# B&R Automation Studio project AriesV2 (part 4)

#### Cyclic.st
```iecst
PROGRAM _CYCLIC

	gRecCfg;
//
//	CASE gHmi.prv.currentPage OF
//		HMI_RECIPE_20_SELECT:
//			pRecCfgUIConnect ACCESS ADR(gRecipe_CSV_UIConnect);
//			pCmd ACCESS ADR(loc.Rec.HMI);
//		HMI_RECIPE_21_PVLIST:
//			pRecCfgUIConnect ACCESS ADR(gRecipe_CSV_UIConnect);
//			pCmd ACCESS ADR(loc.Rec.HMI);
//		HMI_CONFIG_30_SELECT:
//			pRecCfgUIConnect ACCESS ADR(gConfig_CSV_UIConnect);
//			pCmd ACCESS ADR(loc.Cfg.HMI);
//		HMI_CONFIG_31_PVLIST:
//			pRecCfgUIConnect ACCESS ADR(gConfig_CSV_UIConnect);
//			pCmd ACCESS ADR(loc.Cfg.HMI);
//		HMI_LOGIN_43_ENGINEER:
//			pRecCfgUIConnect ACCESS ADR(gConfig_CSV_UIConnect);
//			pCmd ACCESS ADR(loc.Cfg.HMI);
//	END_CASE;
//
//
//	IF EDGENEG(gHmi.prv.currentPage = HMI_RECIPE_20_SELECT) THEN
//		locFindActiveRecipe := 1;
//	END_IF;
//
//	IF EDGENEG(gHmi.prv.currentPage = HMI_CONFIG_30_SELECT) THEN
//		locFindActiveRecipe := 1;
//	END_IF;
//
//	IF loc.Rec.cmd.Copy_default_to_save = 1 THEN
//		gRecCfg.save.Rec := gRecCfg.defaultvals.Rec;
//	END_IF;
//
//	IF loc.Rec.cmd.Copy_default_to_active = 1 THEN
//		gRecCfg.active.Rec := gRecCfg.defaultvals.Rec;
//	END_IF;
//
//	IF loc.Rec.cmd.Copy_save_to_active = 1 THEN
//		gRecCfg.active.Rec := gRecCfg.save.Rec;
//	END_IF;
//
//	IF loc.Rec.cmd.Copy_save_to_default = 1 THEN
//		gRecCfg.defaultvals.Rec := gRecCfg.save.Rec;
//	END_IF;
//
//	IF loc.Rec.cmd.Copy_active_to_save = 1 THEN
//		gRecCfg.save.Rec := gRecCfg.active.Rec;
//	END_IF;
//
//	IF loc.Rec.cmd.Copy_active_to_default = 1 THEN
//		gRecCfg.defaultvals.Rec := gRecCfg.active.Rec;
//	END_IF;
//
//	IF loc.Rec.cmd.Copy_internal_to_default = 1 THEN
////		Set_Default_Rec;
//	END_IF;
//
//	gRecCfg.save.Cfg.Motor.Home := gRecCfg.active.Cfg.Motor.Home;
//
//	loc.Cfg.status.save_differs_from_active := BOOL_TO_USINT(brsmemcmp(ADR(gRecCfg.save.Cfg),ADR(gRecCfg.active.Cfg), SIZEOF(Global_Cfg_typ)) <> 0);
//	loc.Cfg.status.default_differs_from_save := BOOL_TO_USINT(brsmemcmp(ADR(gRecCfg.defaultvals.Cfg),ADR(gRecCfg.save.Cfg), SIZEOF(Global_Cfg_typ)) <> 0);
//	loc.Cfg.status.active_differs_from_default := BOOL_TO_USINT(brsmemcmp(ADR(gRecCfg.active.Cfg),ADR(gRecCfg.defaultvals.Cfg), SIZEOF(Global_Cfg_typ)) <> 0);
//
////	loc.Cfg.status.Invalid := NOT Fcn_Config_Valid(pCfg := ADR(gRecCfg.active.Cfg), pAlarms := ADR(gAlarms));
//
//	loc.Rec.status.save_differs_from_active := BOOL_TO_USINT(brsmemcmp(ADR(gRecCfg.save.Rec),ADR(gRecCfg.active.Rec), SIZEOF(Global_Rec_typ)) <> 0);
//	loc.Rec.status.default_differs_from_save := BOOL_TO_USINT(brsmemcmp(ADR(gRecCfg.defaultvals.Rec),ADR(gRecCfg.save.Rec), SIZEOF(Global_Rec_typ)) <> 0);
//	loc.Rec.status.active_differs_from_default := BOOL_TO_USINT(brsmemcmp(ADR(gRecCfg.active.Rec),ADR(gRecCfg.defaultvals.Rec), SIZEOF(Global_Rec_typ)) <> 0);
//
////	loc.Rec.status.Invalid := NOT Fcn_Recipe_Valid(pRec := ADR(gRecCfg.active.Rec), pAlarms := ADR(gAlarms));
//
//	locCurrentlySelectedRecIsActive := (brsstrcmp(ADR(gRecipe_CSV_UIConnect.Recipe.List.Names[gRecipe_CSV_UIConnect.Recipe.List.SelectedIndex]), ADR(gRecipeName)) = 0);
//	locCurrentlySelectedCfgIsActive := (brsstrcmp(ADR(gConfig_CSV_UIConnect.Recipe.List.Names[gConfig_CSV_UIConnect.Recipe.List.SelectedIndex]), ADR(gConfigName)) = 0);
//
//	CASE pRecCfgUIConnect.MessageBox.Type OF
//		mpRECIPE_UI_MSG_CONFIRM_LOAD:
//
//		mpRECIPE_UI_MSG_CONFIRM_SAVE:
//
//			IF EDGEPOS(pRecCfgUIConnect.MessageBox.Confirm) THEN
//				CASE gHmi.prv.currentPage OF
//					HMI_RECIPE_20_SELECT:
//						gRecCfg.save.Rec := gRecCfg.active.Rec;
//					HMI_CONFIG_30_SELECT:
//						gRecCfg.save.Cfg := gRecCfg.active.Cfg;
//				END_CASE;
//			END_IF;
//		mpRECIPE_UI_MSG_CONFIRM_CREATE:
//
//		mpRECIPE_UI_MSG_CONFIRM_DELETE:
//			CASE gHmi.prv.currentPage OF
//				HMI_RECIPE_20_SELECT:
//					IF EDGEPOS(gRecipe_CSV_UIConnect.MessageBox.Confirm) THEN
//						IF (brsstrcmp(ADR(gRecipe_CSV_UIConnect.Recipe.List.Names[gRecipe_CSV_UIConnect.Recipe.List.SelectedIndex]), ADR(gRecipeName)) = 0) THEN
//							gRecipe_CSV_UIConnect.MessageBox.Confirm := FALSE; //can't delete active recipe
//							gRecipe_CSV_UIConnect.MessageBox.Cancel := TRUE;
//						END_IF;
//					END_IF;
//				HMI_CONFIG_30_SELECT:
//					IF EDGEPOS(gConfig_CSV_UIConnect.MessageBox.Confirm) THEN
//						IF (brsstrcmp(ADR(gConfig_CSV_UIConnect.Recipe.List.Names[gConfig_CSV_UIConnect.Recipe.List.SelectedIndex]), ADR(gConfigName)) = 0) THEN
//							gConfig_CSV_UIConnect.MessageBox.Confirm := FALSE; //can't delete active recipe
//							gConfig_CSV_UIConnect.MessageBox.Cancel := TRUE;
//						END_IF;
//					END_IF;
//			END_CASE;
//	END_CASE;
//	//
//	IF loc.Rec.HMI.Refresh.DP = 1 THEN
//		gRecipe_CSV_UIConnect.Recipe.Refresh := 1;
//	END_IF;
//
//	IF loc.Cfg.HMI.Refresh.DP = 1 THEN
//		gConfig_CSV_UIConnect.Recipe.Refresh := 1;
//	END_IF;
//
//	loc.Rec.HMI.Refresh.DP := 0;
//	loc.Rec.HMI.Refresh.Status := DINT_TO_BOOL(gHmiParamTable.selValueFormVisible = 1);
//	loc.Rec.HMI.Refresh.Lock := 0;
//
//	loc.Cfg.HMI.Refresh.DP := 0;
//	//
//	IF loc.Rec.HMI.Save.DP = 1 THEN
//
//		//Make sure listbox selected recipe name is the active one when you are trying to save from a page other than the Rec/Cfg control page (Saving on PVListView page)
//		Action_Set_Active_Rec;
//
//		gRecipe_CSV_UIConnect.Recipe.Save := 1;
//	END_IF;
//
//	IF loc.Cfg.HMI.Save.DP = 1 THEN
//		gConfig_CSV_UIConnect.Recipe.Save := 1;
//	END_IF;
//	//
//	loc.Rec.HMI.Save.DP := 0;
//	loc.Rec.HMI.Save.Status := NOT (loc.Rec.status.save_differs_from_active = 1) OR ((NOT (locCurrentlySelectedRecIsActive = 1)) AND gHmi.prv.currentPage = HMI_RECIPE_21_PVLIST) OR DINT_TO_BOOL(gHmiParamTable.selValueFormVisible = 1);
//	loc.Rec.HMI.Save.Lock := 0;
//
//	loc.Cfg.HMI.Save.DP := 0;
//
//	//
//	IF loc.Rec.HMI.Load.DP = 1 THEN
//		gRecipe_CSV_UIConnect.Recipe.Load := 1;
//	END_IF;
//
//	IF loc.Cfg.HMI.Load.DP = 1 THEN
//		gConfig_CSV_UIConnect.Recipe.Load := 1;
//	END_IF;
//	//
//	loc.Rec.HMI.Load.DP := 0;
//	loc.Rec.HMI.Load.Status :=  DINT_TO_BOOL(gHmiParamTable.selValueFormVisible = 1);
//	loc.Rec.HMI.Load.Lock := 0;
//
//	loc.Cfg.HMI.Load.DP := 0;
//	//
//	IF loc.Rec.HMI.Delete.DP = 1 THEN
//		gRecipe_CSV_UIConnect.Recipe.Delete := 1;
//	END_IF;
//
//	IF loc.Cfg.HMI.Delete.DP = 1 THEN
//		gConfig_CSV_UIConnect.Recipe.Delete := 1;
//	END_IF;
//	//
//	loc.Rec.HMI.Delete.DP := 0;
//	loc.Rec.HMI.Delete.Status := locCurrentlySelectedRecIsActive OR DINT_TO_BOOL(gHmiParamTable.selValueFormVisible = 1);
//	loc.Rec.HMI.Delete.Lock := 0;
//
//	loc.Cfg.HMI.Delete.DP := 0;
//	//
//	IF loc.Rec.HMI.Overwrite.DP = 1 THEN
//		gRecCfg.IO.Rec.I.FileName := gRecipe_CSV_UIConnect.Recipe.List.Names[gRecipe_CSV_UIConnect.Recipe.List.SelectedIndex];
//		Recipe_CSV_Control.Save := TRUE;
//	END_IF;
//
//	IF loc.Cfg.HMI.Overwrite.DP = 1 THEN
//		gRecCfg.IO.Cfg.I.FileName := gConfig_CSV_UIConnect.Recipe.List.Names[gConfig_CSV_UIConnect.Recipe.List.SelectedIndex];
//		Config_CSV_Control.Save := TRUE;
//	END_IF;
//	//
//	loc.Rec.HMI.Overwrite.DP := 0;
//	//	loc.Rec.HMI.Overwrite.Status := locCurrentlySelectedRecIsActive OR DINT_TO_BOOL(gHmiParamTable.selValueFormVisible = 1);
//	loc.Rec.HMI.Overwrite.Status := 1;
//	loc.Rec.HMI.Overwrite.Lock := 0;
//
//	IF loc.Rec.HMI.Copy.DP = 1 THEN
//		locDTGetTime.enable := 1;
//		locDTGetTime();
//		locTimeString := '';
//		ascDT(locDTGetTime.DT1, ADR(locTimeString), 255);
//		gRecCfg.IO.Rec.I.FileName := '';
//		gRecCfg.IO.Rec.I.FileName := gRecipeName;
//		brsmemset(ADR(gRecCfg.IO.Rec.I.FileName) + brsstrlen(ADR(gRecCfg.IO.Rec.I.FileName)) - 4, 0,1);
//		brsstrcat(ADR(gRecCfg.IO.Rec.I.FileName), ADR('_cpy_'));
//		brsstrcat(ADR(gRecCfg.IO.Rec.I.FileName), ADR(locTimeString));
//		brsstrcat(ADR(gRecCfg.IO.Rec.I.FileName), ADR('.csv'));
//		FOR ii_char := 0 TO brsstrlen(ADR(gRecCfg.IO.Rec.I.FileName)) BY 1 DO
//			IF brsmemcmp(ADR(gRecCfg.IO.Rec.I.FileName) + ii_char, ADR(':'), 1) = 0 OR brsmemcmp(ADR(gRecCfg.IO.Rec.I.FileName) + ii_char, ADR(' '), 1) = 0 THEN
//				brsmemset(ADR(gRecCfg.IO.Rec.I.FileName) + ii_char, 95, 1);
//			END_IF;
//		END_FOR;
//		Recipe_CSV_Control.Save := 1;
//	END_IF;
//
//	loc.Rec.HMI.Copy.DP := 0;
//	loc.Rec.HMI.Copy.Status := NOT (locCurrentlySelectedRecIsActive = 1) OR DINT_TO_BOOL(gHmiParamTable.selValueFormVisible = 1);
//	loc.Rec.HMI.Copy.Lock := 0;
//
//	loc.Cfg.HMI.Refresh.Status := DINT_TO_BOOL(gHmiParamTable.selValueFormVisible = 1);
//	loc.Cfg.HMI.Save.Status := DINT_TO_BOOL(gHmiParamTable.selValueFormVisible = 1);
//	loc.Cfg.HMI.Load.Status := DINT_TO_BOOL(gHmiParamTable.selValueFormVisible = 1);
//	loc.Cfg.HMI.Delete.Status := DINT_TO_BOOL(gHmiParamTable.selValueFormVisible = 1);
//	loc.Cfg.HMI.Overwrite.Status := 1;
//	loc.Cfg.HMI.Copy.Status := 1;
//
//	locRefreshBeforeCall := gRecipe_CSV_UIConnect.Recipe.Refresh;
//
//	Recipe_CSV_Control;
//	Recipe_CSV_RegPar;
//	Recipe_CSV_UI;
//	pRecCfgUIConnect;
//	gRecipe_CSV_UIConnect;
//
//	Config_CSV_Control;
//	Config_CSV_RegPar;
//	Config_CSV_UI;
//	gConfig_CSV_UIConnect;
//
//	IF (NOT gRecipe_CSV_UIConnect.Recipe.Refresh AND locRefreshBeforeCall) OR locFindActiveRecipe = 1 THEN
//		bgTimerStart(loc_Timer_Find_Active, Tms(0.5));
//		locFindActiveRecipe := 0;
//	END_IF;
//
////	IF EDGEPOS(bgTimerIsTimeOut(loc_Timer_Find_Active)) THEN
////		FOR ii_recipes := 0 TO 19 BY 1 DO
////			IF (brsstrcmp(ADR(gRecipe_CSV_UIConnect.Recipe.List.Names[ii_recipes]), ADR(gRecipeName)) = 0) THEN
////				gRecipe_CSV_UIConnect.Recipe.List.SelectedIndex := ii_recipes;
////			END_IF;
////		END_FOR;
//	//	END_IF;
//
//	IF EDGEPOS(bgTimerIsTimeOut(loc_Timer_Find_Active)) THEN
//		Action_Set_Active_Rec;
//	END_IF;
//	//
//	IF Recipe_CSV_Control.CommandDone AND (Recipe_CSV_Control.Save OR Recipe_CSV_Control.Load) THEN
//		Recipe_CSV_Control.Save := FALSE;
//		Recipe_CSV_Control.Load := FALSE;
//		gRecipe_CSV_UIConnect.Recipe.Refresh := 1;
//	END_IF;
//
//	IF EDGENEG(gRecipe_CSV_UIConnect.Status = mpRECIPE_UI_STATUS_SAVE) THEN
////		gRecipeName := Recipe_CSV_Control.Info.LastLoadedRecipe;
//		gRecCfg.save.Rec := gRecCfg.active.Rec;
//	END_IF;
//
//	IF EDGENEG(gRecipe_CSV_UIConnect.Status = mpRECIPE_UI_STATUS_LOAD) THEN
//		gRecipeName := Recipe_CSV_Control.Info.LastLoadedRecipe;
//		gRecCfg.active.Rec := gRecCfg.save.Rec;
//	END_IF;
//
//	loc.Rec.cmd.Copy_default_to_save := FALSE;
//	loc.Rec.cmd.Copy_default_to_active := FALSE;
//	loc.Rec.cmd.Copy_save_to_active := FALSE;
//	loc.Rec.cmd.Copy_save_to_default := FALSE;
//	loc.Rec.cmd.Copy_active_to_save := FALSE;
//	loc.Rec.cmd.Copy_active_to_default := FALSE;
//	loc.Rec.cmd.Copy_internal_to_default := FALSE;
//
//	bgTimerCyclic(loc_Timer_Find_Active);
//	//
//
//	IF Config_CSV_Control.CommandDone AND (Config_CSV_Control.Save OR Config_CSV_Control.Load) THEN
//		Config_CSV_Control.Save := FALSE;
//		Config_CSV_Control.Load := FALSE;
//		gConfig_CSV_UIConnect.Recipe.Refresh := 1;
//	END_IF;
//
//	IF EDGENEG(gConfig_CSV_UIConnect.Status = mpRECIPE_UI_STATUS_SAVE) THEN
////		gConfigName := Config_CSV_Control.Info.LastLoadedRecipe;
//		gRecCfg.save.Cfg := gRecCfg.active.Cfg;
//	END_IF;
//
//	IF EDGENEG(gConfig_CSV_UIConnect.Status = mpRECIPE_UI_STATUS_LOAD) THEN
//		gConfigName := Config_CSV_Control.Info.LastLoadedRecipe;
//		gRecCfg.active.Cfg := gRecCfg.save.Cfg;
//	END_IF;
//
//	loc.Cfg.cmd.Copy_default_to_save := FALSE;
//	loc.Cfg.cmd.Copy_default_to_active := FALSE;
//	loc.Cfg.cmd.Copy_save_to_active := FALSE;
//	loc.Cfg.cmd.Copy_save_to_default := FALSE;
//	loc.Cfg.cmd.Copy_active_to_save := FALSE;
//	loc.Cfg.cmd.Copy_active_to_default := FALSE;
//	loc.Cfg.cmd.Copy_internal_to_default := FALSE;
//	//
END_PROGRAM
```

### Program Logical/pkgAlert/AlarmX (IEC)

#### Main.st - Init, cyclic, exit code
```iecst
PROGRAM _INIT
	(* Insert code here *)
	AlarmX_Control.MpLink := ADR(MpLink_AlarmControl);
	AlarmX_Control.Enable := TRUE;

	AlarmX_ListUI.MpLink := ADR(MpLink_AlarmControl);
	AlarmX_ListUI.Enable := TRUE;
	AlarmX_ListUI.UISetup.AlarmListSize := 5;
	AlarmX_ListUI.UISetup.AlarmListScrollWindow := 5;
	AlarmX_ListUI.UIConnect := ADR(AlarmX_ListUIConnect);

	AlarmX_History.MpLink := ADR(MpLink_AlarmHistory);
	AlarmX_History.Enable := TRUE;
	AlarmX_History.DeviceName := ADR('Alarm');
	AlarmX_History.Language := ADR('en');

	AlarmX_HistoryUI.MpLink := ADR(MpLink_AlarmHistory);
	AlarmX_HistoryUI.Enable := TRUE;
	AlarmX_HistoryUI.UISetup.AlarmListSize := 5;
	AlarmX_HistoryUI.UISetup.AlarmListScrollWindow := 5;
	AlarmX_HistoryUI.UIConnect := ADR(AlarmX_History_UIConnect);

//	AlarmX_ListUIConnect.AlarmList.Timestamp[0]

END_PROGRAM

PROGRAM _CYCLIC

	IF set THEN
		set := FALSE;
		MpAlarmXSet(MpLink_AlarmControl, 'exampleAlarm');
	END_IF;

	IF reset THEN
		reset := FALSE;
		MpAlarmXReset(MpLink_AlarmControl, 'exampleAlarm');
	END_IF;

	IF ack THEN
		ack := FALSE;
		MpAlarmXAcknowledge(MpLink_AlarmControl, 'exampleAlarm');
	END_IF;

	loc.ExampleAlarm.active := MpAlarmXCheckState(MpLink_AlarmControl, 'exampleAlarm', mpALARMX_STATE_NONE);
	loc.ExampleReaction.active := MpAlarmXCheckReaction(MpLink_AlarmControl, 'exampleReaction');

	AlarmX_Control();
	AlarmX_ListUI();
	AlarmX_ListUIConnect;

	AlarmX_History();
	AlarmX_HistoryUI();
	AlarmX_History_UIConnect;
END_PROGRAM

PROGRAM _EXIT
	(* Insert code here *)

END_PROGRAM
```

#### Variables.var - Local variables
```iecst
VAR
	reset : BOOL;
	set : BOOL;
	ack : BOOL;
	loc : AlarmX_Local_TmpVar_typ;
END_VAR
```

### Program Logical/pkgAlert/ComLogger

#### Cyclic.st
```iecst
PROGRAM _CYCLIC
	Com_Logger_UI;
	Com_Logger_UIConnect;
END_PROGRAM
```

#### Init.st
```iecst
PROGRAM _INIT
	Com_Logger_UI.Enable := TRUE;

//	Com_Logger_UI.MpLink := ADR(mpCOM_MAIN);

	Com_Logger_UI.Scope := mpCOM_CONFIG_SCOPE_BRANCH;

	Com_Logger_UI.UISetup.LoggerListSize := 8;
	Com_Logger_UI.UISetup.LoggerScrollWindow := 1;

	Com_Logger_UI.UIConnect := ADR(Com_Logger_UIConnect);

	Com_Logger_UI;
	Com_Logger_UIConnect;
END_PROGRAM
```

### Data_Global.var
```iecst
VAR
	File_Manager_Control : MpFileManagerUI := (0);
	File_Manager_UIConnect : MpFileManagerUIConnectType := (0);
END_VAR
```

### Program Logical/pkgData/File_Handling (IEC)

#### Cyclic.st
```iecst
PROGRAM _CYCLIC
	File_Manager_Control;
	File_Manager_UIConnect;
END_PROGRAM
```

### Program Logical/pkgData/DataTask

#### Main.st
```iecst
PROGRAM _INIT
	Data_Log_Control.MpLink := ADR(Data_Log_MpLink);
	Data_Log_Control.Enable := TRUE;
	Data_Log_Control.Header := ADR(Data_Log_Header);
	Data_Log_Control.DeviceName := ADR('Data_Log');
//	Data_Log_Control.RecordMode := mpDATA_RECORD_MODE_TRIGGER;
	Data_Log_Control.RecordMode := mpDATA_RECORD_MODE_TIME;
	Data_Log_Control.Record := TRUE;
	Data_Log_Control();
//
	Data_Table_Control.MpLink := ADR(Data_Log_MpLink);
	Data_Table_Control.Enable := TRUE;
	Data_Table_Control.UISetup.ValueListSize := 10;
	Data_Table_Control.UISetup.ValueListScrollWindow := 1;
	Data_Table_Control.UISetup.PVListSize := 5;
	Data_Table_Control.UISetup.PVListScrollWindow := 1;
	Data_Table_Control.UIConnect := ADR(Data_Table_UIConnect);
	Data_Table_Control();
	Data_Table_UIConnect;

END_PROGRAM

PROGRAM _CYCLIC
	Data_Log_Control.Record := TRUE;
//	Data_Log_Control.SamplingTime := Tms(gRecCfg.active.Cfg.Mechanics.T_Record_Data_S);
//	Data_Log_Control.SamplingTime := Tms(600); //TODO: Change back

	Data_Log_Config;
	Data_Log_Config_Struct;
	Data_Log_Control;
	Data_Log_Header;
	Data_Log_RegPar;

	Data_Log_Control.Trigger := FALSE;

	Data_Table_Control();
	Data_Table_UIConnect;

END_PROGRAM

PROGRAM _EXIT
	(* Insert code here *)

END_PROGRAM
```

### pvListView_Global_Var.var
```iecst
VAR
	gTableStats : hmiTableStats_typ;
END_VAR
```

### Program Logical/pkgPVListView/HMITableManager (IEC)

#### Variables.var - Local variables
```iecst
VAR
	loc : HMITableControlLocal_typ;
	Init_Logbook : FBK_Init_Logbook;
	tmp_bool : BOOL;
END_VAR
```

### Library Logical/pkgPVListView/paiPVTable

#### HMIparamList.typ
```iecst
(********************************************************************
 * COPYRIGHT -- piedmont
 ********************************************************************
 * Package: HMI
 * File: HMI.typ
 * Author: goran
 * Created: August 28, 2013
 ********************************************************************
 * Data types of package HMI
 ********************************************************************)
(*########################################################################*)
(*HMI object - PARAMETER LIST - LIMITS*)
(*########################################################################*)
(*########################################################################*)
(*HMI object - PARAMETER LIST*)
(*########################################################################*)

TYPE
	hmiTableStatStruct_typ : 	STRUCT
		maxLenDesc : UDINT;
		maxLenName : UDINT;
		Param : UDINT;
		Default : UDINT;
		Min : UDINT;
		Max : UDINT;
		Hide : UDINT;
	END_STRUCT;
	hmiTableStats_typ : 	STRUCT
		Overall : hmiTableStatStruct_typ;
	END_STRUCT;
	PVList_Language_Texts_typ : 	STRUCT
		PVTextLangSpecific : STRING[DEFINE_PAR_NAME_MAXLEN];
		PVDescLangSpecific : STRING[DEFINE_PAR_DESC_MAXLEN];
	END_STRUCT;
	PVListTexts_Info_typ : 	STRUCT
		Str : STRING[DEFINE_PAR_NAME_MAXLEN];
		isValid : BOOL;
		isPV : BOOL;
		isConstant : BOOL;
		Const_Value : REAL;
		PVAdr : {REDUND_UNREPLICABLE} UDINT;
		PVLen : USINT;
		PVDim : USINT;
		PVTyp : UDINT;
		StrLen : UDINT;
	END_STRUCT;
	PVTable_Val_Info_typ : 	STRUCT
		Param : PVListTexts_Info_typ;
		Default : PVListTexts_Info_typ;
		Min : PVListTexts_Info_typ;
		Max : PVListTexts_Info_typ;
		Hide : PVListTexts_Info_typ;
	END_STRUCT;
	PVTableInfo : 	STRUCT
		PVText : ARRAY[0..MAX_IDX_LANGUAGES]OF PVList_Language_Texts_typ;
		Val : PVTable_Val_Info_typ;
		Error : BOOL;
	END_STRUCT;
	HMI_Table_Data_typ : 	STRUCT
		info : ARRAY[0..DEFINE_MAX_TABLE_ENTRIES]OF PVTableInfo;
		Max_Idx_Entries : UDINT;
		Table_Name : STRING[DEFINE_PAR_NAME_MAXLEN];
		NameSpace : STRING[DEFINE_PAR_NAME_MAXLEN];
		Load_OK : BOOL;
	END_STRUCT;
	hmiParamLimits_typ : 	STRUCT
		k_factor : REAL; (*scaling k factor (y=kx + n, where y=dsiplay value, x=plc value)*)
		n_factor : REAL; (*scaling n factor (y=kx + n, where y=dsiplay value, x=plc value)*)
		minValue : REAL; (*min value*)
		maxValue : REAL; (*max value*)
		defaultValue : REAL; (*default value*)
		pEnumText : UDINT; (*ptr to a string of comma delimited enum texts*)
		pEnumVals : UDINT; (*ptr to a string of comma delimited enum values*)
		valueType : UINT; (*type of the paramvalue (0-DINT, 1-REAL, 2-ENUM)*)
	END_STRUCT;
	hmiParamListTable_typ : 	STRUCT
		listHeader : STRING[DEFINE_PAR_NAME_MAXLEN]; (*name of the list (header text)*)
		listIdText : ARRAY[0..DEFINE_MAX_TABLE_ENTRIES]OF STRING[DEFINE_PAR_IDX_MAXLEN]; (*table colum: id-s*)
		listTypeText : ARRAY[0..DEFINE_MAX_TABLE_ENTRIES]OF STRING[DEFINE_PAR_NAME_MAXLEN]; (*table colum: value*)
		listDefaultText : ARRAY[0..DEFINE_MAX_TABLE_ENTRIES]OF STRING[DEFINE_PAR_NAME_MAXLEN]; (*table colum: value*)
		listMinText : ARRAY[0..DEFINE_MAX_TABLE_ENTRIES]OF STRING[DEFINE_PAR_NAME_MAXLEN]; (*table colum: value*)
		listMaxText : ARRAY[0..DEFINE_MAX_TABLE_ENTRIES]OF STRING[DEFINE_PAR_NAME_MAXLEN]; (*table colum: value*)
		listValueText : ARRAY[0..DEFINE_MAX_TABLE_ENTRIES]OF STRING[DEFINE_PAR_NAME_MAXLEN]; (*table colum: value*)
		listName : ARRAY[0..DEFINE_MAX_TABLE_ENTRIES]OF STRING[DEFINE_PAR_NAME_MAXLEN]; (*table colum: name*)
		listDescription : ARRAY[0..DEFINE_MAX_TABLE_ENTRIES]OF STRING[DEFINE_PAR_DESC_MAXLEN]; (*table colum: description*)
		listValuePtr : ARRAY[0..DEFINE_MAX_TABLE_ENTRIES]OF UDINT; (*list of ptrs to parametars*)
		listDecPlaces : ARRAY[0..DEFINE_MAX_TABLE_ENTRIES]OF DINT; (*list of dec places for each parametar*)
		listLimits : ARRAY[0..DEFINE_MAX_TABLE_ENTRIES]OF hmiParamLimits_typ;
		selName : {REDUND_UNREPLICABLE} STRING[DEFINE_PAR_NAME_MAXLEN]; (*name of the currently selected/active parametar*)
		selDescription : STRING[DEFINE_PAR_DESC_MAXLEN]; (*description of the currently selected/active parametar*)
		selValueEnumIndex : UDINT; (*value of the currently selected/active parametar for type enum*)
		selValueEnumIndexMax : UDINT; (*value of the currently selected/active parametar for type enum*)
		selValueREAL : REAL; (*value of the currently selected/active parametar*)
		selValueREALOld : REAL; (*value of the currently selected/active parametar (previous value for change detection*)
		selValueREALMax : REAL; (*max value of the currently selected/active parametar*)
		selValueREALMin : REAL; (*min value of the currently selected/active parametar*)
		selValueREALDefault : REAL; (*default value of the currently selected/active parametar*)
		selValueDecPlaces : DINT; (*default value of the currently selected/active parametar*)
		selValueDINT : DINT; (*value of the currently selected/active parametar*)
		selValueDINTOld : DINT; (*value of the currently selected/active parametar (previous value for change detection*)
		selValueDINTMax : DINT; (*max value of the currently selected/active parametar*)
		selValueDINTMin : DINT; (*min value of the currently selected/active parametar*)
		selValueDINTDefault : DINT; (*default value of the currently selected/active parametar*)
		selValueFormVisible : DINT; (*visibility control of the form / controls for setting parametar value*)
		index : UINT; (*index of the currently selected/active parametar*)
		indexOld : UINT; (*index of the currently selected/active parametar (previous value for change detection)*)
		maxIndex : UINT; (*max index / number of items in the table. Must be less then hmiTableMAXDESCRIPTION!!!*)
		setDefaultRequest : BOOL; (*set default request flag*)
		incDP : USINT;
		decDP : USINT;
	END_STRUCT;
END_TYPE
```

#### Constants.var
```iecst
VAR CONSTANT
	MAX_IDX_LANGUAGES : UDINT := 5;
	DEFINE_LANGUAGE_STRINGS : ARRAY[0..MAX_IDX_LANGUAGES] OF STRING[4] := ['en','sv','pt','de','es','fr']; (*MUST MATCH EXACTLY THE LANGUAGES IN THE ORDER THEY ARE CONFIGURED IN PROJECT LANGUAGES.*)
	DEFINE_MAX_IDX_HMI_TABLES : UDINT := 12;
	DEFINE_MAX_TABLE_ENTRIES : UDINT := 18;
	DEFINE_PAR_DESC_MAXLEN : UDINT := 255;
	DEFINE_PAR_NAME_MAXLEN : UDINT := 80;
	DEFINE_PAR_IDX_MAXLEN : UDINT := 4;
	DEFINE_PAR_VALUE_MAXLEN : UDINT := 12;
	DEFINE_INDEX_TEXTTABLE_PV : USINT := 0;
	DEFINE_INDEX_TEXTTABLE_DEFAULT : USINT := 1;
	DEFINE_INDEX_TEXTTABLE_MIN : USINT := 2;
	DEFINE_INDEX_TEXTTABLE_MAX : USINT := 3;
	DEFINE_INDEX_TEXTTABLE_HIDE : USINT := 4;
	DEFINE_LOGSTRING_LEN : UDINT := 200;
END_VAR
(*Insert your comment here.*)
```

#### paiPVTable.fun
```iecst
FUNCTION hmiParamListTableCyclic : USINT
	VAR_INPUT
		p_int : UDINT;
	END_VAR
END_FUNCTION

FUNCTION_BLOCK hmiTableFBK_typ (*TODO: Add your comment here*) (*$GROUP=User,$CAT=User,$GROUPICON=User.png,$CATICON=User.png*)
	VAR_INPUT
		tableName : STRING[DEFINE_PAR_NAME_MAXLEN];
		nameSpace : STRING[DEFINE_PAR_NAME_MAXLEN];
		hmiStruct : {REDUND_UNREPLICABLE} HMI_Table_Data_typ;
		Logbook : UDINT;
		TableStats : {REDUND_UNREPLICABLE} hmiTableStatStruct_typ;
		pOverallStats : REFERENCE TO hmiTableStatStruct_typ;
	END_VAR
END_FUNCTION_BLOCK

FUNCTION ActivateHMITable : BOOL (*TODO: Add your comment here*) (*$GROUP=User,$CAT=User,$GROUPICON=User.png,$CATICON=User.png*)
	VAR_INPUT
		langIdx : DINT;
		pHMITable : UDINT;
		pTableValues : UDINT;
	END_VAR
END_FUNCTION
```

#### ActivateHMITable.c
```c
#include <bur/plctypes.h>
#ifdef __cplusplus
	extern "C"
	{
#endif
	#include "paiPVTable.h"
#ifdef __cplusplus
	};
#endif
#include "hmiParamList.h"
#include "ArTextSys.h"
/* TODO: Add your comment here */

REAL PVStructInfo(PVListTexts_Info_typ * p){

	UDINT val_int = 0;
	REAL val_real = 0;

	if(!p || !(p->isValid)){
		return 0;
	}else if(p->isConstant){
		return p->Const_Value;
	}

	switch(p->PVTyp){
		case 7: //UDINT
			val_int = *((UDINT *)(p->PVAdr));
			val_real = (REAL) val_int;
			break;
		case 8: //REAL
			val_real = *((REAL * )(p->PVAdr));
			break;
	}

	return val_real;

}

plcbit ActivateHMITable(DINT langIdx, UDINT pHMITable_int, UDINT pTableValues_int)
{
	hmiParamListTable_typ * pHMITable = pHMITable_int;
	HMI_Table_Data_typ * pTableValues = pTableValues_int;
	UDINT ii_entries = 0;
	UINT valtype;
	DINT dec_places;
	REAL val_min;
	REAL val_max;
	REAL val_def;
	UDINT * val_hide_int;

	BOOL val_hide_bool = 0;

	if(pTableValues->Max_Idx_Entries >= DEFINE_MAX_TABLE_ENTRIES) return 0;

	hmiParamListTableEntryFirst(pHMITable, (char *) &pTableValues->Table_Name);
	for(ii_entries = 0; ii_entries <= pTableValues->Max_Idx_Entries; ii_entries++){
		if(pTableValues->info[ii_entries].Val.Hide.isValid==1){
			val_hide_int = ((UDINT *) (pTableValues->info[ii_entries].Val.Hide.PVAdr));
			val_hide_bool = (BOOL) (*val_hide_int);
		}else{
			val_hide_bool = 0;
		}

		if(val_hide_bool==0 && pTableValues->info[ii_entries].Val.Param.PVAdr){
			val_min = PVStructInfo(&pTableValues->info[ii_entries].Val.Min);
			val_max = PVStructInfo(&pTableValues->info[ii_entries].Val.Max);
			val_def = PVStructInfo(&pTableValues->info[ii_entries].Val.Default);

				switch(pTableValues->info[ii_entries].Val.Param.PVTyp){
					case 7: //UDINT
						valtype=0;
						dec_places=-2; //no decimals
						break;
					case 8: //REAL
						valtype=1;
						dec_places=1;
						break;
				}

				hmiParamListTableAddEntryNext(pHMITable,
					pTableValues->info[ii_entries].Val.Param.PVAdr,
					&pTableValues->info[ii_entries].PVText[langIdx].PVTextLangSpecific,
					val_def,val_min,val_max,
					dec_places,1,0,valtype,
					&pTableValues->info[ii_entries].PVText[langIdx].PVDescLangSpecific
					);
			}
		}
	hmiParamListTableEntryLast(pHMITable);
}
```

#### hmiTableFBK_typ.c
```c
/// IAUTOMATION CONFIDENTIAL
/// Unpublished Copyright (c) 2016 iAutomation, All Rights Reserved.
///
/// NOTICE:  All information contained herein is, and remains the property of iAutomation. The intellectual and technical concepts contained
/// herein are proprietary to iAutomation and may be covered by U.S. and Foreign Patents, patents in process, and are protected by trade secret or copyright law.
/// Dissemination of this information or reproduction of this material is strictly forbidden unless prior written permission is obtained
/// from iAutomation.  Access to the source code contained herein is hereby forbidden to anyone except current iAutomation employees, managers or contractors who have executed
/// Confidentiality and Non-disclosure agreements explicitly covering such access.
///
/// The copyright notice above does not evidence any actual or intended publication or disclosure  of  this source code, which includes
/// information that is confidential and/or proprietary, and is a trade secret, of  iAutomation.   ANY REPRODUCTION, MODIFICATION, DISTRIBUTION, PUBLIC  PERFORMANCE,
/// OR PUBLIC DISPLAY OF OR THROUGH USE  OF THIS  SOURCE CODE  WITHOUT  THE EXPRESS WRITTEN CONSENT OF COMPANY IS STRICTLY PROHIBITED, AND IN VIOLATION OF APPLICABLE
/// LAWS AND INTERNATIONAL TREATIES.  THE RECEIPT OR POSSESSION OF  THIS SOURCE CODE AND/OR RELATED INFORMATION DOES NOT CONVEY OR IMPLY ANY RIGHTS
/// TO REPRODUCE, DISCLOSE OR DISTRIBUTE ITS CONTENTS, OR TO MANUFACTURE, USE, OR SELL ANYTHING THAT IT  MAY DESCRIBE, IN WHOLE OR IN PART.
///
/// Programmer: John C. Glisson
/// Date: 20. October 2016

#include <bur/plctypes.h>
#ifdef __cplusplus
	extern "C"
	{
#endif
	#include "paiPVTable.h"
#ifdef __cplusplus
	};
#endif

#include "hmiParamList.h"
#include "ArTextSys.h"

static void Update_Stats_Table(UDINT * pMaxVal, char * pText, UDINT * pOverallMaxVal){
	UDINT TextLen = 0;

	TextLen = brsstrlen((UDINT) pText);

	if(*pMaxVal < TextLen){
		*pMaxVal = TextLen;
	}
	if(*pOverallMaxVal < TextLen){
		*pOverallMaxVal = TextLen;
	}
	return;
}

static DINT writeText(char * pNameSpace, char * pText, char * pLangCode, char * pParName, UDINT Buffer_Size, UDINT * pTextLen){
	STRING Buffer[Buffer_Size];
	ArTextSysGetText_typ FBK;
	FBK.Namespace = (UDINT) pNameSpace;
	FBK.SearchMode = arTEXTSYS_SEARCH_LANGUAGE_ONLY;
	FBK.TextID = (UDINT) pText;
	brsstrcpy((UDINT) &FBK.LanguageCode, (UDINT) pLangCode);
	FBK.TextBuffer =(UDINT) &Buffer;
	FBK.TextBufferSize = Buffer_Size;

	FBK.Execute = 0;
	ArTextSysGetText(&FBK);
	FBK.Execute = 1;
	ArTextSysGetText(&FBK);

	if(FBK.StatusID == 0){
		brsstrcpy((UDINT) pParName, (UDINT) &Buffer);
		*pTextLen = brsstrlen((UDINT) &Buffer);
	}else{
		brsstrcpy((UDINT) pParName,(UDINT)  &"Err");
	}
	return FBK.StatusID;
}

static DINT Get_PV_Table_Item_Info(char * pNameSpace, char * pTextID, char * pLangCode, PVListTexts_Info_typ * p){
	DINT status = 0;

	status = writeText(pNameSpace,pTextID,pLangCode,(char *) &p->Str, DEFINE_PAR_NAME_MAXLEN, &p->StrLen);

	if(status==0){
		p->isValid = 1;
	}else{
		p->isValid = 0;
		return status;
	}

	status = PV_xgetadr((UDINT) &p->Str,(UDINT) &p->PVAdr,(UDINT) &p->PVLen);

	if(status==0){
		p->isPV = 1;
		p->isConstant = 0;
	}else{
		p->isPV = 0;
		p->isConstant = 1;
		p->Const_Value = brsatof((UDINT) &p->Str);
		return status;
	}

	status = PV_ninfo((UDINT) &p->Str,(UDINT) &p->PVTyp,(UDINT) &p->PVLen,(UDINT) &p->PVDim);
	return status;
}

static void GetPVTableInfo(char * pNameSpace, UDINT pvTableIdx, PVTableInfo * p, BOOL * pErrorFlag){
	char strPVID[DEFINE_PAR_NAME_MAXLEN] = "PV.";
	char strPVIdx[DEFINE_PAR_IDX_MAXLEN];
	DINT status = 0;

	brsitoa(pvTableIdx,(UDINT)  &strPVIdx);
	brsstrcat((UDINT) &strPVID, (UDINT) &strPVIdx);

	status = Get_PV_Table_Item_Info(pNameSpace,		(char *) &strPVID,		(char *) &DEFINE_LANGUAGE_STRINGS[DEFINE_INDEX_TEXTTABLE_PV], 		&p->Val.Param);
	status = Get_PV_Table_Item_Info(pNameSpace,		(char *) &strPVID,		(char *) &DEFINE_LANGUAGE_STRINGS[DEFINE_INDEX_TEXTTABLE_MIN], 		&p->Val.Min);
	status = Get_PV_Table_Item_Info(pNameSpace,		(char *) &strPVID,		(char *) &DEFINE_LANGUAGE_STRINGS[DEFINE_INDEX_TEXTTABLE_MAX], 		&p->Val.Max);
	status = Get_PV_Table_Item_Info(pNameSpace,		(char *) &strPVID,		(char *) &DEFINE_LANGUAGE_STRINGS[DEFINE_INDEX_TEXTTABLE_DEFAULT], 	&p->Val.Default);
	status = Get_PV_Table_Item_Info(pNameSpace,		(char *) &strPVID,		(char *) &DEFINE_LANGUAGE_STRINGS[DEFINE_INDEX_TEXTTABLE_HIDE], 	&p->Val.Hide);
	return;
}

static void GetPVNameInfo(char * pNameSpace, UDINT idxLanguage, UDINT idxPV, char * pParName, char * pParDesc, BOOL * pErrorFlag){
	ArTextSysLanguageCodeType strTmpLang;
	brsstrcpy((UDINT) &strTmpLang, (UDINT) &DEFINE_LANGUAGE_STRINGS[idxLanguage]);
	char strPVName[DEFINE_PAR_NAME_MAXLEN] = "Title.";
	char strPVDesc[DEFINE_PAR_DESC_MAXLEN] = "Desc.";
	char strPVIdx[DEFINE_PAR_IDX_MAXLEN];
	brsitoa((DINT) idxPV, (UDINT) &strPVIdx);
	brsstrcat((UDINT) &strPVName, (UDINT) &strPVIdx);
	brsstrcat((UDINT) &strPVDesc, (UDINT) &strPVIdx);
	UDINT TextLen = 0;

	writeText(pNameSpace, (char *) &strPVName, (char *) &strTmpLang, pParName, DEFINE_PAR_NAME_MAXLEN, &TextLen);
	writeText(pNameSpace, (char *) &strPVDesc, (char *) &strTmpLang, pParDesc, DEFINE_PAR_DESC_MAXLEN, &TextLen);
}

void hmiTableFBK_typ(struct hmiTableFBK_typ* p)
{
	//Really going to try hard to do this all in one cycle.
	UDINT ii_entries=0;
	UDINT ii_languages=0;

	BOOL flagError = 0;

	STRING LogString[DEFINE_LOGSTRING_LEN];

	brsstrcpy((UDINT) &p->hmiStruct.Table_Name,(UDINT)  &p->tableName);
	brsstrcpy((UDINT) &p->hmiStruct.NameSpace,(UDINT)  &p->nameSpace);

	for(ii_entries = 0; ii_entries <= DEFINE_MAX_TABLE_ENTRIES; ii_entries++){
		GetPVTableInfo(p->nameSpace, ii_entries, &p->hmiStruct.info[ii_entries], &flagError);

		if(p->hmiStruct.info[ii_entries].Val.Param.PVAdr == 0){//If there isn't a PV at that index, return from the function...
			p->hmiStruct.Max_Idx_Entries = ii_entries - 1;
			p->hmiStruct.Load_OK = (flagError == 0);

			wbrsnprintf((char *) &LogString, DEFINE_LOGSTRING_LEN, "TableInfo:<Table=%s><Count=%d><err=%d>", &p->tableName, ii_entries, (UDINT) flagError);
			requestMessageToLog((char *) &LogString, p->Logbook, arlogLEVEL_INFO, 50000, 0, 0);

			return;
		}//...Otherwise load its texts

		wbrsnprintf((char *) &LogString, DEFINE_LOGSTRING_LEN, "TableItem:<PVName=%s><Def=%s><Min=%s><Max=%s>", &p->hmiStruct.info[ii_entries].Val.Param.Str, &p->hmiStruct.info[ii_entries].Val.Default.Str, &p->hmiStruct.info[ii_entries].Val.Min.Str, &p->hmiStruct.info[ii_entries].Val.Max.Str);
		requestMessageToLog((char *) &LogString, p->Logbook, arlogLEVEL_INFO, 50000, 0, 0);

		Update_Stats_Table(&p->TableStats.Param,(char *) &p->hmiStruct.info[ii_entries].Val.Param.Str, &p->pOverallStats->Param);
		Update_Stats_Table(&p->TableStats.Default,(char *) &p->hmiStruct.info[ii_entries].Val.Default.Str, &p->pOverallStats->Default);
		Update_Stats_Table(&p->TableStats.Min,(char *) &p->hmiStruct.info[ii_entries].Val.Min.Str, &p->pOverallStats->Min);
		Update_Stats_Table(&p->TableStats.Max,(char *) &p->hmiStruct.info[ii_entries].Val.Max.Str, &p->pOverallStats->Max);
		Update_Stats_Table(&p->TableStats.Hide,(char *) &p->hmiStruct.info[ii_entries].Val.Hide.Str, &p->pOverallStats->Hide);

		for(ii_languages = 0; ii_languages <= MAX_IDX_LANGUAGES; ii_languages++){
			GetPVNameInfo((char *) &p->nameSpace, ii_languages, ii_entries,(char *) &p->hmiStruct.info[ii_entries].PVText[ii_languages].PVTextLangSpecific,(char *)  &p->hmiStruct.info[ii_entries].PVText[ii_languages].PVDescLangSpecific, &flagError);

			Update_Stats_Table(&p->TableStats.maxLenDesc,(char *) &p->hmiStruct.info[ii_entries].PVText[ii_languages].PVDescLangSpecific, &p->pOverallStats->maxLenDesc);
			Update_Stats_Table(&p->TableStats.maxLenName,(char *) &p->hmiStruct.info[ii_entries].PVText[ii_languages].PVTextLangSpecific, &p->pOverallStats->maxLenName);
		}
	}
}
```

### Enumerations.typ
```iecst
TYPE
	HERNON_Dispense_Enum :
		(
		DISPENSE_STATE_INIT := 0,
		DISPENSE_STATE_READY := 1,
		DISPENSE_STATE_DISPENSING := 2,
		DISPENSE_STATE_WAIT_RESET := 3,
		DISPENSE_STATE_INACTIVE := 4,
		DISPENSE_STATE_DISABLED := 5,
		DISPENSE_STATE_ERROR := 6,
		DISPENSE_STATE_WAIT_ADDITIONAL := 8,
		STATE_WAIT_FRACTION_OFFSET := 9
		);
	HERNON_DISP_REASONS_ENUM :
		(
		DISPENSE_SINGLE_SHOT := 0,
		DISPENSE_PURGE := 1
		);
END_TYPE
```

### RecCfgParams.typ
```iecst
(*Insert your comment here.*)

TYPE
	HERNON_Cfg_Dispense_typ : 	STRUCT
		Disable : UDINT;
	END_STRUCT;
	HERNON_Rec_Dispense_typ : 	STRUCT
		Enable : UDINT;
		Disp_Valve_Edgemode_Pulse_TO_ms : REAL;
		Fractional_Position_Offset : REAL;
		Extra_Shots_Per_VBlock : UDINT;
		Time_Offset_Additional_Shots : REAL;
		Target_Offset : UDINT;
	END_STRUCT;
END_TYPE

(*Insert your comment here.*)
```

### Program Logical/Application/Master/ControlLogic (IEC)

#### Action_Dispense_TriggerFinger.st
```iecst
ACTION Action_Dispense_TriggerFinger:
	IF Position.Current_Target <> Position_LastCycle.Current_Target THEN
		FOR ii_valves := 0 TO MAX_IDX_VALVES BY 1 DO
			IF gRecCfg.active.Cfg.Dispense[ii_valves].Disable = 0 AND gRecCfg.active.Rec.Dispense[ii_valves].Enable = 1 THEN
				IF TargetInfoArray[Control.Dispense[ii_valves].Current_Target_At_Dispense_Unit].VBlock_Occupied AND NOT TargetInfoArray[Control.Dispense[ii_valves].Current_Target_At_Dispense_Unit].VBlock_Dispensed[ii_valves] THEN
					IF ValveFBK[ii_valves].iFlagDispenseOnFractionOffset THEN
						gStatistics.Debug.Disp_Flag_Twice[ii_valves].Count := gStatistics.Debug.Disp_Flag_Twice[ii_valves].Count + 1;
						gStatistics.Debug.Disp_Flag_Twice[ii_valves].Latch_Position := Position;

					ELSE
						ValveFBK[ii_valves].iFlagDispenseOnFractionOffset := TRUE;
						gStatistics.Debug.Disp_Trigger_Count[ii_valves].Count := gStatistics.Debug.Disp_Trigger_Count[ii_valves].Count + 1;
						TargetInfoArray[Control.Dispense[ii_valves].Current_Target_At_Dispense_Unit].VBlock_Dispensed[ii_valves] := TRUE;
					END_IF;
				END_IF;
			END_IF;
		END_FOR;
	END_IF;
END_ACTION
```

#### Action_Dial_Position_Velocity_Calc.st
```iecst
ACTION Action_Dial_Position_Velocity_Calc:

	IF gRecCfg.active.Cfg.Control.Sim_Encoder = 1 THEN
		Dashboard_Hide_Encoder_Sim := STATUS_LIGHT_FLASH.bFlashOut;
		ii_cycles := ii_cycles + 1;
		IF ii_cycles >= gRecCfg.active.Cfg.Control.Sim_Encoder_Cycles THEN
			ii_cycles := 0;
			sim_encoder := sim_encoder + UDINT_TO_UINT(gRecCfg.active.Cfg.Control.Sim_Encoder_Counts);

			IF sim_encoder > 4095 THEN
				sim_encoder := 0;
			END_IF;
		END_IF;

		gAlarms.Control.Encoder_Sim_Active := TRUE;

		PositionValue := sim_encoder;
	ELSE
		gAlarms.Control.Encoder_Sim_Active := FALSE;
		Dashboard_Hide_Encoder_Sim := 1;
		PositionValue := ControlIO.iEncoderValue;
	END_IF;

	ShiftBits := 16 - UDINT_TO_UINT(gRecCfg.active.Cfg.Control.N_Encoder_Bits_SingleTurn);

	//Shift bits left to take advantage of natural 16-bit rollover.  Effectively this is the same as multiplying by 8 for a 12 bit encoder, but it accomodates multiple bit counts (up to 16) and multiturn encoders (shifts multiturn bits "off the end")
	Position_SHL.Single_Turn_Absolute := 		SHL(PositionValue, ShiftBits);
	Position_SHL.Home_Position := 				SHL(UDINT_TO_UINT(gRecCfg.active.Cfg.Control.Encoder_Position_Home), ShiftBits);
	Position_SHL.Single_Turn_Rel_Home := 		Position_SHL.Single_Turn_Absolute - Position_SHL.Home_Position;
	Position_SHL.Ticks_Per_Target := 			REAL_TO_UINT((2**16) / UDINT_TO_REAL(gRecCfg.active.Rec.Control.N_Targets_On_Dial)); //This operation MUST be done like this such that it rounds instead of "floors" which causes swamping drift (where floor is the effective operation when dividing integers!)
	Position_SHL.Current_Target := 				Position_SHL.Single_Turn_Rel_Home / Position_SHL.Ticks_Per_Target;
	Position_SHL.Ticks_Within_Current_Target := Position_SHL.Single_Turn_Rel_Home MOD Position_SHL.Ticks_Per_Target;

	//Shift bits back right
	Position.Single_Turn_Absolute 			:= 		SHR(Position_SHL.Single_Turn_Absolute, ShiftBits);
	Position.Home_Position 					:= 		SHR(Position_SHL.Home_Position, ShiftBits);
	Position.Single_Turn_Rel_Home 			:= 		SHR(Position_SHL.Single_Turn_Rel_Home, ShiftBits);
	Position.Ticks_Per_Target 				:= 		SHR(Position_SHL.Ticks_Per_Target, ShiftBits);
	Position.Current_Target 				:= 		Position_SHL.Current_Target;
	Position.Ticks_Within_Current_Target 	:= 		SHR(Position_SHL.Ticks_Within_Current_Target, ShiftBits);
	Position.Degrees_Absolute				:=		360 * (UINT_TO_REAL(Position.Single_Turn_Absolute) / (2**gRecCfg.active.Cfg.Control.N_Encoder_Bits_SingleTurn));
	Position.Home_Position_Degrees			:=		360 * (UINT_TO_REAL(Position.Home_Position) / (2**gRecCfg.active.Cfg.Control.N_Encoder_Bits_SingleTurn));
	Position.Degrees_Rel_Home				:=		360 * (UINT_TO_REAL(Position.Single_Turn_Rel_Home) / (2**gRecCfg.active.Cfg.Control.N_Encoder_Bits_SingleTurn));
	Position.Target_Fractional_Position_Pct :=		100 * (UINT_TO_REAL(Position.Ticks_Within_Current_Target) / UINT_TO_REAL(Position.Ticks_Per_Target));

	encoder_diff_counts := (SHR((UINT_TO_INT(Position_SHL.Single_Turn_Absolute) - UINT_TO_INT(Position_SHL_LastCycle.Single_Turn_Absolute)), ShiftBits));

	Multiturn_Absolute_Position := Multiturn_Absolute_Position + encoder_diff_counts;

	VelCalc_DT_Element.In := DINT_TO_REAL(Multiturn_Absolute_Position);
	VelCalc_DT_Element();

	Dial_Vel.Encoder_Counts_Per_Second := VelCalc_DT_Element.Out;
	Dial_Vel.Rev_Per_S := Dial_Vel.Encoder_Counts_Per_Second / (2**gRecCfg.active.Cfg.Control.N_Encoder_Bits_SingleTurn);
	Dial_Vel.Targ_Per_S := Dial_Vel.Rev_Per_S * UDINT_TO_REAL(gRecCfg.active.Rec.Control.N_Targets_On_Dial);
	Dial_Vel.Deg_Per_S := Dial_Vel.Rev_Per_S * 360;
	Dial_Vel.RPM := 60 * Dial_Vel.Rev_Per_S;

END_ACTION
```

#### Action_Test_PiP_Trigger.st
```iecst
ACTION Action_Test_PiP_Trigger:
//	//TEST PIP trigger output to sync the encoder position to PIP sensor so I can capture traces on O-Scope RDH
	IF Position.Target_Fractional_Position_Pct > 1 AND Position.Target_Fractional_Position_Pct < 25 THEN
		ControlIO.Inspection.oInspectionGood := 1;
	ELSE
		ControlIO.Inspection.oInspectionGood := 0;
	END_IF

	IF Position.Target_Fractional_Position_Pct > 50 AND Position.Target_Fractional_Position_Pct < 75 THEN
		ControlIO.Inspection.oInspectionValid := 1;
	ELSE
		ControlIO.Inspection.oInspectionValid := 0;
	END_IF
END_ACTION
```

#### Action_HMI_Commands_Handler.st
```iecst
ACTION Action_HMI_Commands_Handler:
	//Command from HMI to reset home position to encoder "0" position->
	IF CMD_Set_Home_Pos_0 THEN
		CMD_Set_Home_Pos_0 := FALSE;
		gRecCfg.active.Cfg.Control.Encoder_Position_Home := 0;
	END_IF;

	//Command from HMI to set home position as current encoder position->
	IF CMD_Set_Current_Pos_As_Home THEN
		CMD_Set_Current_Pos_As_Home := FALSE;
		gRecCfg.active.Cfg.Control.Encoder_Position_Home := Position.Single_Turn_Absolute;
	END_IF;

	//Command from HMI to reset stats counters->
	IF CMD_Reset_Statistics THEN
		CMD_Reset_Statistics := FALSE;
		brsmemset(ADR(gStatistics), 0, SIZEOF(AS3500HS_Stats_typ));
	END_IF;
END_ACTION
```

### Library Logical/Application/Master/libAS52XX (IEC)
Depends on: AsBrStr

#### Enumerations.typ
```iecst
TYPE
	HERNON_AS_Prcs_HMI_Colors_Enum :
		(
		HMI_PRCS_COLOR_DISABLED := 0,
		HMI_PRCS_COLOR_IDLE := 1,
		HMI_PRCS_COLOR_ACTIVE := 2,
		HMI_PRCS_COLOR_FAULT := 3
		);
END_TYPE
```

### Program Logical/Auxiliary_Services_Control/ComLogger

#### Cyclic.st
```iecst
PROGRAM _CYCLIC
	Com_Logger_UI;
	Com_Logger_UIConnect;

	gMachineName;
	gProjectDate;
	gVersion;
END_PROGRAM
```

### Program Logical/pkgAccess/UserX

#### Main.st
```iecst
PROGRAM _INIT

END_PROGRAM

PROGRAM _CYCLIC

END_PROGRAM

PROGRAM _EXIT
	(* Insert code here *)

END_PROGRAM
```

### HTMLVis.typ
```iecst
TYPE
	HTML_Alert_typ : 	STRUCT
		numAlarms : DINT;
		numWarnings : DINT;
		idxImage : DINT;
		cycle : DINT;
	END_STRUCT;
	HMTLMotionPVs_typ : 	STRUCT
		indexAxis : DINT;
		FBK_Read_Error : MC_ReadAxisError;
		ErrText : STRING[STRLEN_AXIS_ERROR];
	END_STRUCT;
	HTML_ExampleTrend_typ : 	STRUCT
		New_Member2 : USINT;
		New_Member1 : USINT;
		New_Member : USINT;
	END_STRUCT;
	HTMLVis_typ : 	STRUCT
		Motion : HMTLMotionPVs_typ;
		Alert : HTML_Alert_typ;
		Trend : HTML_ExampleTrend_typ;
		New_Member2 : USINT;
		New_Member1 : USINT;
		New_Member : USINT;
	END_STRUCT;
END_TYPE
```

### Program Logical/pkgMpViewAux/VisCtrl (IEC)

#### Types.typ
```iecst
TYPE
	ClientInfo : 	STRUCT
		IpAddress : WSTRING[64];
		UserId : WSTRING[64];
		ActivityCount : UDINT;
		LanguageId : STRING[2];
		MeasurementSystemId : WSTRING[32];
		ConnectionDateTime : DATE_AND_TIME;
		ScreenResolution : WSTRING[16];
		BrowserResolution : WSTRING[16];
		UserAgent : WSTRING[256];
		CookieEnabled : BOOL;
		SlotId : USINT;
		IsValid : BOOL;
	END_STRUCT;
END_TYPE
```

#### Variables.var
```iecst
VAR
	usint_tmp : USINT;
	clientSlots : ARRAY[0..4] OF ClientInfo;
	pAxisControl : REFERENCE TO MpAxisBasic;
	pDelta : REFERENCE TO MpDelta4Axis;
	pAxisPar : REFERENCE TO MpAxisBasicParType;
END_VAR
```

### OEE_Global.var
```iecst
VAR
	OEE_Trend_UIConnect : MpOeeTrendUIConnectType;
	OEE_List_UIConnect : MpOeeListUIConnectType;
	OEE_Core_UIConnect : MpOeeCoreUIConnectType;
	OEE_Timeline_UIConnect : MpOeeTimelineUIConnectType;
END_VAR
```

### Safety_typ.typ
```iecst
TYPE
	paiSL_Operations_typ : 	STRUCT
		Ack_All_UDID : BOOL;
		Ack_Firmware : BOOL;
		Ack_Safekey_Exchange : BOOL;
		Test_LED : BOOL;
		Sys_Scan : BOOL;
		Alter_SK_Password : BOOL;
		Format_SK : BOOL;
		Reset : BOOL;
		Clear_Data : BOOL;
		Download_Application : BOOL;
	END_STRUCT;
	paiSL_Public_In_typ : 	STRUCT
		Password_for_command : STRING[16];
		Password_New : STRING[16];
		Command : paiSL_Operations_typ;
		Reset : BOOL;
	END_STRUCT;
	paiSL_RCTRL_Public_out_typ : 	STRUCT
		Status : paiSafeLogicStatusOut_Enum;
		State : paiSafeLogicStateOut_Enum;
		SafeOSState : paiSafeLogicSafeOSOut_Enum;
		FailSafe : BOOL;
	END_STRUCT;
	paiSL_Public_Out_typ : 	STRUCT
		State : paiInitSafelogicStates_Enum;
		Command_Allowed : paiSL_Operations_typ;
		HMI_Hide : paiSL_Operations_typ;
		Command_Being_Executed : paiSL_Operations_typ;
		Status_Print : STRING[255];
		RCTRL : paiSL_RCTRL_Public_out_typ;
		State_Old : paiInitSafelogicStates_Enum;
	END_STRUCT;
	paiSL_FBK_typ : 	STRUCT
		RemoteControl : safeRemoteControl;
		DownloadApplication : safeDownloadApplication;
		UDID_Low : AsIOAccRead;
		UDID_High : AsIOAccRead;
	END_STRUCT;
	paiSL_Read_UDID_typ : 	STRUCT
		Value : UDINT;
		Valid : BOOL;
	END_STRUCT;
	paiSL_Data_typ : 	STRUCT
		RemoteControlCmd : RemoteControlCmdTypeV1;
		DownloadAppCmd : DownloadCmdApplicationTypeV1;
		Read_UDID_High : paiSL_Read_UDID_typ;
		Read_UDID_Low : paiSL_Read_UDID_typ;
	END_STRUCT;
	paiSL_prv_timers_typ : 	STRUCT
		Timer_Print_HMI_Status : TON;
		Timer_Max_RCTRL_Cmd : TON;
		Timer_Error_Retry : TON;
		Timer_Rescan : TON;
	END_STRUCT;
	paiSL_Prv_typ : 	STRUCT
		FBK : paiSL_FBK_typ;
		Data : paiSL_Data_typ;
		Timer : paiSL_prv_timers_typ;
		Command_Number : UINT;
	END_STRUCT;
	paiSL_typ : 	STRUCT
		i : paiSL_Public_In_typ;
		o : paiSL_Public_Out_typ;
		prv : paiSL_Prv_typ;
	END_STRUCT;
	paiSafeLogicSafeOSOut_Enum :
		(
		SAFEOS_INVALID_OR_BOOT := 0,
		SAFEOS_ON_OR_ERROR := 1,
		SAFEOS_LOADING := 2,
		SAFEOS_STOP_SAFE := 3,
		SAFEOS_RUN_SAFE := 4,
		SAFEOS_HALT_DEBUG := 5,
		SAFEOS_STOP_DEBUG := 6,
		SAFEOS_RUN_DEBUG := 7,
		SAFEOS_NO_EXECUTION := 8,
		SAFEOS_UPDATING_STATUS := 9
		);
	paiSafeLogicStateOut_Enum :
		(
		RCTRL_IDLE := 0,
		RCTRL_ENTER_RECD := 1,
		RCTRL_EXECUTING_ENTER := 2,
		RCTRL_PREPARING_ENTER := 3,
		RCTRL_ENTER_EXECUTED_WAIT_RESET := 4
		);
	paiSafeLogicStatusOut_Enum :
		(
		COMMAND_VALID_IN_EXECUTION := 0,
		HMI_COMMAND_EXECUTE_SUCCESS := 1,
		HMI_COMMAND_EXECUTE_ERROR := 2,
		REMOTE_COMMAND_EXECUTE_SUCCESS := 3,
		REMOTE_COMMAND_EXECUTE_ERROR := 4,
		ERROR_COMMAND_UNKNOWN := 5,
		ERROR_ENTER_COMMAND_UNKNOWN := 6,
		ERROR_RCTRL_DISABLED_SAFEDES := 7,
		ERROR_INCORRECT_PASSWORD := 8,
		ERROR_RCTRL_SM_NOT_IDLE := 9,
		ERROR_LOCKED_AT_HMI := 10,
		ERROR_SW_ACK_UNAUTHORIZED := 11,
		ERROR_FW_ACK_UNAUTHORIZED := 12,
		ERR_SMX_TO_CMX_UNAUTHORIZED := 13,
		ERR_SK_ACK_CANT_EXECUTE := 14,
		FW_ACK_CANT_EXECUTE := 15,
		ERR_SMX_CANT_EXECUTE := 16,
		ERR_DMX_CANT_EXECUTE := 17,
		ERR_TMX_CANT_EXECUTE := 18,
		ERR_QMX_CANT_EXECUTE := 19,
		ERR_CMX_CANT_EXECUTE := 20,
		ERR_SK_CONTINUE_CANT_EXEC := 21,
		ERR_ENTER_IMPOSS_SK_ACK_REQD := 22,
		ERR_SK_FORMAT_EXECUTING_SL_LOCK := 23,
		ERR_SK_COPY_EXECUTING_SL_LOCK := 24,
		ERR_SK_ACK_EXECUTING_SL_LOCK := 25,
		ERR_SMX_ACK_CMX_EXECUTING := 26,
		ERR_SCAN_EXECUTING_SL_LOCK := 27,
		ERR_REMOTE_SEND_FAILURE := 28,
		ERR_INCORRECT_CMD_LEN := 29,
		ERR_INCORRECT_CMD_LEN_2 := 30,
		ERR_USRDATA_FORMAT_RUNNING := 31
		);
	paiInitSafelogicStates_Enum :
		(
		SAFE_PROGRAM_INIT := 0,
		SAFE_PROGRAM_READ_STATUS := 1,
		SAFE_PROGRAM_WAIT_COMMAND := 2,
		SAFE_PROGRAM_DOWNLOAD_APP := 4,
		SAFE_PROGRAM_SET_PASSWORD := 5,
		SAFE_PROGRAM_FORMAT_SAFEKEY := 6,
		SAFE_PROGRAM_CONFIRM_SK_XCHG := 7,
		SAFE_PROGRAM_CONFIRM_FW := 8,
		SAFE_PROGRAM_SCAN := 9,
		SAFE_PROGRAM_LED_TEST := 10,
		SAFE_PROGRAM_CLEAR_DATA := 11,
		SAFE_PROGRAM_CONFIRM_MODULES := 12,
		SAFE_PROGRAM_RESET := 14,
		SAFE_PROGRAM_ERROR := 15,
		SAFE_PROGRAM_PRINT_STATUS_WAIT := 16,
		SAFE_PROGRAM_READ_UDID := 17
		);
	paiSL_Perm_Info_typ : 	STRUCT
		Safekey_Formatted : USINT;
		Password_Set : USINT;
		Application_Downloaded : USINT;
		SKey_Exchanged : USINT;
		ACK_UDID_Firmware : USINT;
		Run_State : USINT;
	END_STRUCT;
END_TYPE
```

### Program Logical/pkgSafety/SafeINIT (IEC)

#### Action_Init_RCTRL_Cmd.st
```iecst
ACTION Action_Init_RCTRL_Cmd:
	brsmemset(ADR(gSafety.o.Command_Allowed), 0, SIZEOF(paiSL_Operations_typ));
	brsmemset(ADR(gSafety.o.Command_Being_Executed), 0, SIZEOF(paiSL_Operations_typ));

	gSafety.prv.FBK.DownloadApplication.Execute := FALSE;
	gSafety.prv.FBK.UDID_High.enable := FALSE;
	gSafety.prv.FBK.UDID_Low.enable := FALSE;

	gSafety.o.RCTRL.SafeOSState := SAFEOS_UPDATING_STATUS;
	gSafety.prv.Data.RemoteControlCmd.Password := gSafety.i.Password_for_command;
	gSafety.prv.Data.RemoteControlCmd.NewPassword := '';
	gSafety.prv.Command_Number := gSafety.prv.Command_Number + 1;
	gSafety.prv.Data.RemoteControlCmd.Number := gSafety.prv.Command_Number;
	gSafety.prv.Data.RemoteControlCmd.Command := safeCMD_ENTER;
	gSafety.prv.FBK.RemoteControl.Execute := TRUE;

	bgTimerStart(gSafety.prv.Timer.Timer_Max_RCTRL_Cmd, Tms(DEFINE_TIME_MAX_RCTRL_CMD));
END_ACTION
```

#### Main.st
```iecst
PROGRAM _INIT
//	Init_Logbook.Enable := TRUE;
//	Init_Logbook.Name := 'usr_safe';
//	Init_Logbook();

	gSafety.o.State := SAFE_PROGRAM_INIT;

	gSafety.prv.FBK.RemoteControl.SafeLOGICID := DEFINE_SAFELOGIC_ID;
	gSafety.prv.FBK.RemoteControl.pCommandData := ADR(gSafety.prv.Data.RemoteControlCmd);
	gSafety.prv.Data.RemoteControlCmd.Version := DEFINE_VERSION;

	gSafety.prv.FBK.DownloadApplication.SafeLOGICID := DEFINE_SAFELOGIC_ID;
	gSafety.prv.FBK.DownloadApplication.pCommandData := ADR(gSafety.prv.Data.DownloadAppCmd);
	gSafety.prv.Data.DownloadAppCmd.Version := DEFINE_VERSION;

	gSafety.prv.Command_Number := 0;

	Action_Reset_FBK;
END_PROGRAM

PROGRAM _CYCLIC
	gSafetyPermInfo;

	IF gSafety.i.Reset THEN
		gSafety.i.Reset := FALSE;
		gSafety.o.State := SAFE_PROGRAM_INIT;
	END_IF;

	IF EDGEPOS(gSafety.o.State = SAFE_PROGRAM_WAIT_COMMAND) THEN
		bgTimerStart(gSafety.prv.Timer.Timer_Rescan, Tms(DEFINE_TIME_SCANNING_RETRY));
	END_IF;

	IF EDGEPOS(gSafety.o.State = SAFE_PROGRAM_ERROR) THEN
		bgTimerStart(gSafety.prv.Timer.Timer_Error_Retry, Tms(DEFINE_TIME_ERROR_AUTORESET));
	END_IF;

	IF EDGENEG(gSafety.o.State = SAFE_PROGRAM_WAIT_COMMAND) THEN
		brsmemset(ADR(gSafety.i.Command), 0, SIZEOF(paiSL_Operations_typ));
	END_IF;

	IF EDGEPOS(gSafety.o.State = SAFE_PROGRAM_PRINT_STATUS_WAIT) THEN
		bgTimerStart(gSafety.prv.Timer.Timer_Print_HMI_Status, Tms(DEFINE_TIME_PRINT_HMI_STATUS));
	END_IF;

	//	IF gSafety.o.State <> gSafety.o.State_Old THEN
	//		Data_Log_Control.Trigger := TRUE;
	//	END_IF;

	CASE gSafety.o.State OF
		SAFE_PROGRAM_INIT:
			brsmemset(ADR(gSafety.o.Command_Allowed), 0, SIZEOF(paiSL_Operations_typ));
			Action_Reset_FBK;
			gSafety.o.Status_Print := 'Initializing SL Comm Setup, Please Wait';
			gSafety.o.State := SAFE_PROGRAM_PRINT_STATUS_WAIT;

		SAFE_PROGRAM_READ_STATUS:
			gSafety.prv.Data.RemoteControlCmd.Command := safeCMD_STATUS;
			gSafety.prv.Data.RemoteControlCmd.Data := 0; //Just read the status, data is 0 here per help file

			gSafety.o.Status_Print := 'Reading SafeLogic PLC Status, Please Wait';

			IF gSafety.prv.FBK.RemoteControl.Done AND NOT gSafety.prv.FBK.RemoteControl.Error THEN
				gSafety.o.RCTRL.Status := UINT_TO_DINT(gSafety.prv.FBK.RemoteControl.SafeLOGICStatus.Status);
				gSafety.o.RCTRL.State := UINT_TO_DINT(gSafety.prv.FBK.RemoteControl.SafeLOGICStatus.State);

				CASE gSafety.prv.FBK.RemoteControl.SafeLOGICStatus.SafeOSState OF
					16#00:
					gSafety.o.RCTRL.SafeOSState := SAFEOS_INVALID_OR_BOOT;
					16#0F:
					gSafety.o.RCTRL.SafeOSState := SAFEOS_ON_OR_ERROR;
					//requestMessageToLog(ADR('SafeOS State: On or Error'), Init_Logbook.pLog, arlogLEVEL_INFO,DEFINE_OFFSET_ERR_START + gSafety.prv.Command_Number,0,0);
					16#33:
					gSafety.o.RCTRL.SafeOSState := SAFEOS_LOADING;
					//requestMessageToLog(ADR('SafeOS State: Loading'), Init_Logbook.pLog, arlogLEVEL_INFO,DEFINE_OFFSET_ERR_START + gSafety.prv.Command_Number,0,0);
					16#55:
					gSafety.o.RCTRL.SafeOSState := SAFEOS_STOP_SAFE;
					//requestMessageToLog(ADR('SafeOS State: Stop [Safe]'), Init_Logbook.pLog, arlogLEVEL_INFO,DEFINE_OFFSET_ERR_START + gSafety.prv.Command_Number,0,0);
					16#66:
					gSafety.o.RCTRL.SafeOSState := SAFEOS_RUN_SAFE;
					gSafetyPermInfo.Run_State := 1;
					//requestMessageToLog(ADR('SafeOS State: Run [SAFE]'), Init_Logbook.pLog, arlogLEVEL_INFO,DEFINE_OFFSET_ERR_START + gSafety.prv.Command_Number,0,0);
//					perm_Sys_Commissioned := TRUE;
					16#99:
					gSafety.o.RCTRL.SafeOSState := SAFEOS_HALT_DEBUG;
					//requestMessageToLog(ADR('SafeOS State: Halt [Debug]'), Init_Logbook.pLog, arlogLEVEL_INFO,DEFINE_OFFSET_ERR_START + gSafety.prv.Command_Number,0,0);
					16#AA:
					gSafety.o.RCTRL.SafeOSState := SAFEOS_STOP_DEBUG;
					//requestMessageToLog(ADR('SafeOS State: Stop [Debug]'), Init_Logbook.pLog, arlogLEVEL_INFO,DEFINE_OFFSET_ERR_START + gSafety.prv.Command_Number,0,0);
					16#CC:
					gSafety.o.RCTRL.SafeOSState := SAFEOS_RUN_DEBUG;
					//requestMessageToLog(ADR('SafeOS State: Run [Debug]'), Init_Logbook.pLog, arlogLEVEL_INFO,DEFINE_OFFSET_ERR_START + gSafety.prv.Command_Number,0,0);
					16#F0:
					gSafety.o.RCTRL.SafeOSState := SAFEOS_NO_EXECUTION;
					//requestMessageToLog(ADR('SafeOS State: No Execution'), Init_Logbook.pLog, arlogLEVEL_INFO,DEFINE_OFFSET_ERR_START + gSafety.prv.Command_Number,0,0);
				END_CASE;

				gSafety.o.Command_Allowed.Ack_All_UDID := (gSafety.prv.FBK.RemoteControl.SafeLOGICStatus.NumberOfUDIDMismatches > 0);
				gSafety.o.Command_Allowed.Ack_Firmware := (gSafety.prv.FBK.RemoteControl.SafeLOGICStatus.NumberOfDifferentFirmware > 0);
				gSafety.o.Command_Allowed.Ack_Safekey_Exchange := (gSafety.prv.FBK.RemoteControl.SafeLOGICStatus.SafeKEYChanged > 0);
				gSafety.o.Command_Allowed.Test_LED := TRUE;
				gSafety.o.Command_Allowed.Sys_Scan := TRUE;
				gSafety.o.Command_Allowed.Alter_SK_Password := TRUE;
				gSafety.o.Command_Allowed.Format_SK := TRUE;
				gSafety.o.Command_Allowed.Reset := TRUE;
				gSafety.o.Command_Allowed.Clear_Data := TRUE;
				gSafety.o.Command_Allowed.Download_Application := TRUE;

				gSafety.o.RCTRL.FailSafe := (gSafety.prv.FBK.RemoteControl.SafeLOGICStatus.FailSafe = 16#55);

				gSafety.o.State := SAFE_PROGRAM_WAIT_COMMAND;
			ELSIF gSafety.prv.FBK.RemoteControl.Error AND gSafety.prv.FBK.RemoteControl.StatusID <> 36105 AND gSafety.prv.FBK.RemoteControl.StatusID <> 65535 THEN
				gSafety.o.Status_Print := 'Unable to read status';
				//requestMessageToLog(ADR('Error, RCTRL, attempting to read status'), Init_Logbook.pLog, arlogLEVEL_WARNING,DEFINE_OFFSET_ERR_START + gSafety.prv.FBK.RemoteControl.StatusID,0,0);
				gSafety.o.State := SAFE_PROGRAM_ERROR;
			ELSIF gSafety.prv.FBK.RemoteControl.Error AND gSafety.prv.FBK.RemoteControl.StatusID = 36105 THEN
				gSafety.o.Status_Print := 'Comm Err (Rebooting?)';
				bgTimerStart(gSafety.prv.Timer.Timer_Print_HMI_Status, Tms(DEFINE_TIME_PRINT_HMI_STATUS));
				gSafety.o.State := SAFE_PROGRAM_PRINT_STATUS_WAIT;
			ELSIF bgTimerIsTimeOut(gSafety.prv.Timer.Timer_Max_RCTRL_Cmd) THEN
				gSafety.o.Status_Print := 'Timeout reading status (PLC &| SLX Reboot may be required)';
				//requestMessageToLog(ADR('Status read timeout'), Init_Logbook.pLog, arlogLEVEL_WARNING,gSafety.prv.FBK.RemoteControl.StatusID,0,0);
				gSafety.o.State := SAFE_PROGRAM_ERROR;
			END_IF;

		SAFE_PROGRAM_WAIT_COMMAND:
			Action_Reset_FBK;
			gSafety.o.Status_Print := 'Waiting on User Input Command';

			IF gSafety.prv.FBK.RemoteControl.SafeLOGICStatus.Scanning = 1 AND bgTimerIsTimeOut(gSafety.prv.Timer.Timer_Rescan) AND (gSafety.o.RCTRL.SafeOSState <> SAFEOS_RUN_SAFE) THEN
				gSafety.o.Status_Print := 'Updating SLX status information, please wait';
				gSafety.o.RCTRL.SafeOSState := SAFEOS_UPDATING_STATUS;
				gSafety.o.State := SAFE_PROGRAM_PRINT_STATUS_WAIT;
			ELSIF gSafety.i.Command.Ack_All_UDID THEN
				Action_Init_RCTRL_Cmd;

				CASE gSafety.prv.FBK.RemoteControl.SafeLOGICStatus.NumberOfUDIDMismatches OF
					0:
						gSafety.prv.Data.RemoteControlCmd.Data := safeCMD_1_UDID_ACKN;
					1:
						gSafety.prv.Data.RemoteControlCmd.Data := safeCMD_1_UDID_ACKN;
					2:
						gSafety.prv.Data.RemoteControlCmd.Data := safeCMD_2_UDID_ACKN;
					3:
						gSafety.prv.Data.RemoteControlCmd.Data := safeCMD_3_UDID_ACKN;
					4:
						gSafety.prv.Data.RemoteControlCmd.Data := safeCMD_4_UDID_ACKN;
					ELSE
						gSafety.prv.Data.RemoteControlCmd.Data := safeCMD_N_UDID_ACKN;
				END_CASE;

				//requestMessageToLog(ADR('Acknowledging modules'), Init_Logbook.pLog, arlogLEVEL_INFO,DEFINE_OFFSET_ERR_START + gSafety.prv.Command_Number,0,0);
				gSafety.o.State := SAFE_PROGRAM_CONFIRM_MODULES;
			ELSIF gSafety.i.Command.Ack_Firmware THEN
				Action_Init_RCTRL_Cmd;
				gSafety.prv.Data.RemoteControlCmd.Data := safeCMD_FW_ACKN;
				//requestMessageToLog(ADR('Confirming Firmware'), Init_Logbook.pLog, arlogLEVEL_INFO,DEFINE_OFFSET_ERR_START + gSafety.prv.Command_Number,0,0);
				gSafety.o.State := SAFE_PROGRAM_CONFIRM_FW;
			ELSIF gSafety.i.Command.Ack_Safekey_Exchange THEN
				Action_Init_RCTRL_Cmd;
				gSafety.prv.Data.RemoteControlCmd.Data := safeCMD_SK_XCHG;
				//requestMessageToLog(ADR('Confirming SK Xchg'), Init_Logbook.pLog, arlogLEVEL_INFO,DEFINE_OFFSET_ERR_START + gSafety.prv.Command_Number,0,0);
				gSafety.o.State := SAFE_PROGRAM_CONFIRM_SK_XCHG;
			ELSIF gSafety.i.Command.Test_LED THEN
				Action_Init_RCTRL_Cmd;
				gSafety.prv.Data.RemoteControlCmd.Data := safeCMD_TEST;
				//requestMessageToLog(ADR('Testing LEDs'), Init_Logbook.pLog, arlogLEVEL_INFO,DEFINE_OFFSET_ERR_START + gSafety.prv.Command_Number,0,0);
				gSafety.o.State := SAFE_PROGRAM_LED_TEST;
			ELSIF gSafety.i.Command.Sys_Scan THEN
				Action_Init_RCTRL_Cmd;
				gSafety.prv.Data.RemoteControlCmd.Data := safeCMD_SCAN;
				//requestMessageToLog(ADR('Scanning system...'), Init_Logbook.pLog, arlogLEVEL_INFO,DEFINE_OFFSET_ERR_START + gSafety.prv.Command_Number,0,0);
				gSafety.o.State := SAFE_PROGRAM_SCAN;
			ELSIF gSafety.i.Command.Alter_SK_Password THEN
//				perm_Sys_Commissioned := FALSE;
				Action_Init_RCTRL_Cmd;
				gSafety.prv.Data.RemoteControlCmd.Data := safeCMD_SK_PW;
				gSafety.prv.Data.RemoteControlCmd.NewPassword := gSafety.i.Password_New;
				//requestMessageToLog(ADR('Altering SK password'), Init_Logbook.pLog, arlogLEVEL_INFO,DEFINE_OFFSET_ERR_START + gSafety.prv.Command_Number,0,0);
				gSafety.o.State := SAFE_PROGRAM_SET_PASSWORD;
			ELSIF gSafety.i.Command.Format_SK THEN
				//				perm_Sys_Commissioned := FALSE;
				brsmemset(ADR(gSafetyPermInfo), 0, SIZEOF(paiSL_Perm_Info_typ));
				Action_Init_RCTRL_Cmd;
				gSafety.prv.Data.RemoteControlCmd.Data := safeCMD_SK_FORMAT;
				//requestMessageToLog(ADR('Formatting SafeKey'), Init_Logbook.pLog, arlogLEVEL_INFO,DEFINE_OFFSET_ERR_START + gSafety.prv.Command_Number,0,0);
				gSafety.o.State := SAFE_PROGRAM_FORMAT_SAFEKEY;
			ELSIF gSafety.i.Command.Reset THEN
				Action_Init_RCTRL_Cmd;
				gSafety.prv.Data.RemoteControlCmd.Data := safeCMD_RESET;
				//requestMessageToLog(ADR('Resetting...'), Init_Logbook.pLog, arlogLEVEL_INFO,DEFINE_OFFSET_ERR_START + gSafety.prv.Command_Number,0,0);
				gSafety.o.State := SAFE_PROGRAM_RESET;
			ELSIF gSafety.i.Command.Clear_Data THEN
				Action_Init_RCTRL_Cmd;
				gSafety.prv.Data.RemoteControlCmd.Data := safeCMD_CLEAR_DATA;
				//requestMessageToLog(ADR('Clearing Data'), Init_Logbook.pLog, arlogLEVEL_INFO,DEFINE_OFFSET_ERR_START + gSafety.prv.Command_Number,0,0);
				gSafety.o.State := SAFE_PROGRAM_CLEAR_DATA;
			ELSIF gSafety.i.Command.Download_Application THEN
				gSafety.o.RCTRL.SafeOSState := SAFEOS_UPDATING_STATUS;
				brsmemset(ADR(gSafety.o.Command_Allowed), 0, SIZEOF(paiSL_Operations_typ));
				brsmemset(ADR(gSafety.o.Command_Being_Executed), 0, SIZEOF(paiSL_Operations_typ));
				gSafety.prv.FBK.DownloadApplication.Execute := FALSE;
				gSafety.prv.FBK.RemoteControl.Execute := FALSE;

				gSafety.prv.Data.Read_UDID_Low.Value := 0;
				gSafety.prv.Data.Read_UDID_Low.Valid := FALSE;

				gSafety.prv.Data.Read_UDID_High.Value := 0;
				gSafety.prv.Data.Read_UDID_High.Valid := FALSE;

				gSafety.prv.Data.DownloadAppCmd.Password := gSafety.i.Password_for_command;

				gSafety.prv.Data.DownloadAppCmd.ApplicationID := DEFINE_SAFETY_APP_ID;//TODO: optional functionality not implemented to load .swt file from declared file dev.

				gSafety.prv.FBK.UDID_Low.enable := TRUE;
				gSafety.prv.FBK.UDID_Low.pDeviceName := ADR(DEFINE_SAFELOGIC_ADDRESS);
				gSafety.prv.FBK.UDID_Low.pChannelName := ADR('UDID_low');
				gSafety.prv.FBK.UDID_High.enable := TRUE;
				gSafety.prv.FBK.UDID_High.pDeviceName := ADR(DEFINE_SAFELOGIC_ADDRESS);
				gSafety.prv.FBK.UDID_High.pChannelName := ADR('UDID_high');

				//requestMessageToLog(ADR('Reading UDIDs'), Init_Logbook.pLog, arlogLEVEL_INFO,0,0,0);
				bgTimerStart(gSafety.prv.Timer.Timer_Max_RCTRL_Cmd, Tms(DEFINE_TIME_MAX_RCTRL_CMD));
				gSafety.o.State := SAFE_PROGRAM_READ_UDID;
			END_IF;

		SAFE_PROGRAM_READ_UDID:
			gSafety.o.Status_Print := 'Reading Module UDIDs, please wait';

			IF gSafety.prv.FBK.UDID_Low.status = 0 AND NOT gSafety.prv.Data.Read_UDID_Low.Valid THEN
				gSafety.prv.FBK.UDID_Low.enable := FALSE;
				gSafety.prv.Data.Read_UDID_Low.Value := gSafety.prv.FBK.UDID_Low.value;
				gSafety.prv.Data.Read_UDID_Low.Valid := TRUE;
			END_IF;

			IF gSafety.prv.FBK.UDID_High.status = 0 AND NOT gSafety.prv.Data.Read_UDID_High.Valid THEN
				gSafety.prv.FBK.UDID_High.enable := FALSE;
				gSafety.prv.Data.Read_UDID_High.Value := gSafety.prv.FBK.UDID_High.value;
				gSafety.prv.Data.Read_UDID_High.Valid := TRUE;
			END_IF;

			IF gSafety.prv.Data.Read_UDID_Low.Valid AND gSafety.prv.Data.Read_UDID_High.Valid THEN
				gSafety.prv.Data.DownloadAppCmd.UDID_Low := gSafety.prv.Data.Read_UDID_Low.Value;
				gSafety.prv.Data.DownloadAppCmd.UDID_High := UDINT_TO_UINT(gSafety.prv.Data.Read_UDID_High.Value);

				gSafety.prv.FBK.DownloadApplication.Execute := TRUE;

				gSafety.prv.Data.DownloadAppCmd.Unlock := 0;

				//requestMessageToLog(ADR('UDID Read successful'), Init_Logbook.pLog, arlogLEVEL_INFO,0,0,0);
				bgTimerStart(gSafety.prv.Timer.Timer_Max_RCTRL_Cmd, Tms(DEFINE_TIME_MAX_RCTRL_CMD));
				gSafety.o.State := SAFE_PROGRAM_DOWNLOAD_APP;
			ELSIF gSafety.prv.FBK.UDID_Low.status <> 0 AND gSafety.prv.FBK.UDID_Low.status <> 65535 AND gSafety.prv.FBK.UDID_Low.status <> 65534 AND gSafety.prv.FBK.UDID_High.status <> 0 AND gSafety.prv.FBK.UDID_High.status <> 65535 AND gSafety.prv.FBK.UDID_High.status <> 65534 THEN

				//requestMessageToLog(ADR('UDID Read Error-High'), Init_Logbook.pLog, arlogLEVEL_WARNING,UINT_TO_UDINT(gSafety.prv.FBK.UDID_High.status),0,0);
				//requestMessageToLog(ADR('UDID Read Error-Low'), Init_Logbook.pLog, arlogLEVEL_WARNING,UINT_TO_UDINT(gSafety.prv.FBK.UDID_Low.status),0,0);

				gSafety.o.Status_Print := 'Err reading UDIDs';

				gSafety.o.State := SAFE_PROGRAM_ERROR;
			ELSIF bgTimerIsTimeOut(gSafety.prv.Timer.Timer_Max_RCTRL_Cmd) AND NOT (gSafety.prv.Data.Read_UDID_Low.Valid AND gSafety.prv.Data.Read_UDID_High.Valid) THEN
				gSafety.o.Status_Print := 'Timeout reading UDIDs';
				//requestMessageToLog(ADR('Timeout during UDID Read'), Init_Logbook.pLog, arlogLEVEL_WARNING,0,0,0);
				gSafety.o.State := SAFE_PROGRAM_ERROR;
			END_IF;

		SAFE_PROGRAM_DOWNLOAD_APP:
			gSafety.o.Status_Print := 'Downloading Application from PLC to SafeLogic Controller';

			IF gSafety.prv.FBK.DownloadApplication.UnlockRequired THEN
				gSafety.prv.Data.DownloadAppCmd.Unlock := 1;
			END_IF;

			IF gSafety.prv.FBK.DownloadApplication.Done AND NOT gSafety.prv.FBK.DownloadApplication.Error THEN
				IF gSafety.prv.FBK.DownloadApplication.Error THEN
					//requestMessageToLog(ADR('Error Downloading Application (Did you set the password?)'), Init_Logbook.pLog, arlogLEVEL_WARNING,gSafety.prv.FBK.DownloadApplication.StatusID,0,0);
					gSafety.o.State := SAFE_PROGRAM_ERROR;
				ELSE
					//requestMessageToLog(ADR('Downloaded Application (PLC Power Cycle Required)'), Init_Logbook.pLog, arlogLEVEL_INFO,0,0,0);
					gSafety.o.Status_Print := 'Successfully downloaded application';
					gSafetyPermInfo.Application_Downloaded := 1;
//					perm_Sys_Commissioned := FALSE;
					gSafety.o.State := SAFE_PROGRAM_PRINT_STATUS_WAIT;
				END_IF;
			ELSIF gSafety.prv.FBK.DownloadApplication.Error AND NOT gSafety.prv.FBK.DownloadApplication.StatusID = 65535 THEN
				gSafety.o.Status_Print := 'Error Downloading Application from PLC to SafeLogic Controller';
				//requestMessageToLog(ADR('Error Downloading Application'), Init_Logbook.pLog, arlogLEVEL_WARNING,gSafety.prv.FBK.DownloadApplication.StatusID,0,0);
				gSafety.o.State := SAFE_PROGRAM_ERROR;
			ELSIF bgTimerIsTimeOut(gSafety.prv.Timer.Timer_Max_RCTRL_Cmd) THEN
				gSafety.o.Status_Print := 'Timeout Downloading Program, try again';
				//requestMessageToLog(ADR('Timeout during prog download'), Init_Logbook.pLog, arlogLEVEL_WARNING,0,0,0);
				gSafety.o.State := SAFE_PROGRAM_ERROR;
			END_IF;

		SAFE_PROGRAM_SET_PASSWORD:
			gSafety.o.Status_Print := 'Setting new SLX password';

			IF gSafety.prv.FBK.RemoteControl.Done AND NOT gSafety.prv.FBK.RemoteControl.Error THEN
				IF gSafety.prv.FBK.RemoteControl.Error THEN
					//requestMessageToLog(ADR('Error Altering SLX Password'), Init_Logbook.pLog, arlogLEVEL_WARNING,gSafety.prv.FBK.RemoteControl.StatusID,0,0);
					gSafety.o.State := SAFE_PROGRAM_ERROR;
				ELSE
					//requestMessageToLog(ADR('Changed Password'), Init_Logbook.pLog, arlogLEVEL_INFO,DEFINE_OFFSET_ERR_START + gSafety.prv.Command_Number,0,0);
//					perm_Sys_Commissioned := FALSE;
					gSafety.o.Status_Print := 'Successfully Changed SLX Password';
					gSafetyPermInfo.Password_Set := 1;
					gSafety.o.State := SAFE_PROGRAM_PRINT_STATUS_WAIT;
				END_IF;
			ELSIF gSafety.prv.FBK.RemoteControl.Error THEN
				gSafety.o.Status_Print := 'Error Altering SLX Password';
				//requestMessageToLog(ADR('Error Altering SLX Password'), Init_Logbook.pLog, arlogLEVEL_WARNING,gSafety.prv.FBK.RemoteControl.StatusID,0,0);
				gSafety.o.State := SAFE_PROGRAM_ERROR;
			ELSIF bgTimerIsTimeOut(gSafety.prv.Timer.Timer_Max_RCTRL_Cmd) THEN
				gSafety.o.Status_Print := 'Timeout changing password';
				//requestMessageToLog(ADR('Timeout during password change'), Init_Logbook.pLog, arlogLEVEL_WARNING,DEFINE_OFFSET_ERR_START + gSafety.prv.Command_Number,0,0);
				gSafety.o.State := SAFE_PROGRAM_ERROR;
			END_IF;

		SAFE_PROGRAM_FORMAT_SAFEKEY:
			gSafety.o.Status_Print := 'Formatting Safekey Then Rebooting...';

			IF gSafety.prv.FBK.RemoteControl.Done AND NOT gSafety.prv.FBK.RemoteControl.Error THEN
				IF gSafety.prv.FBK.RemoteControl.Error THEN
					//requestMessageToLog(ADR('Error Formatting Safekey1'), Init_Logbook.pLog, arlogLEVEL_WARNING,gSafety.prv.FBK.RemoteControl.StatusID,0,0);
					gSafety.o.State := SAFE_PROGRAM_ERROR;
				ELSE
					//requestMessageToLog(ADR('Formatted Safekey (Reset required)'), Init_Logbook.pLog, arlogLEVEL_INFO,DEFINE_OFFSET_ERR_START + gSafety.prv.Command_Number,0,0);
//					perm_Sys_Commissioned := FALSE;
					gSafety.o.Status_Print := 'Successfully Formatted Safekey';
					gSafetyPermInfo.Safekey_Formatted := 1;
					bgTimerStart(gSafety.prv.Timer.Timer_Print_HMI_Status, Tms(DEFINE_TIME_PRINT_HMI_STATUS));
					SYSreset(1,1);
					gSafety.o.State := SAFE_PROGRAM_PRINT_STATUS_WAIT;
				END_IF;
			ELSIF gSafety.prv.FBK.RemoteControl.Error AND gSafety.prv.FBK.RemoteControl.StatusID <> 65535 THEN
				gSafety.o.Status_Print := 'Possible error Formatting Safekey (New password?  Powercycle PLC & SLX?)';
				gSafetyPermInfo.Safekey_Formatted := 1;
				//requestMessageToLog(ADR('Error Formatting Safekey2'), Init_Logbook.pLog, arlogLEVEL_WARNING,gSafety.prv.FBK.RemoteControl.StatusID,0,0);
				gSafety.o.State := SAFE_PROGRAM_ERROR;
			ELSIF bgTimerIsTimeOut(gSafety.prv.Timer.Timer_Max_RCTRL_Cmd) THEN
				gSafety.o.Status_Print := 'Timeout formatting SK';
				//requestMessageToLog(ADR('Timeout during SK Format'), Init_Logbook.pLog, arlogLEVEL_WARNING,DEFINE_OFFSET_ERR_START + gSafety.prv.Command_Number,0,0);
				gSafety.o.State := SAFE_PROGRAM_ERROR;
			END_IF;

		SAFE_PROGRAM_CONFIRM_SK_XCHG:
			gSafety.o.Status_Print := 'Confirming Safekey exchange';

			IF gSafety.prv.FBK.RemoteControl.Done AND NOT gSafety.prv.FBK.RemoteControl.Error THEN
				IF gSafety.prv.FBK.RemoteControl.Error THEN
					//requestMessageToLog(ADR('Error during confirming SK XCHG'), Init_Logbook.pLog, arlogLEVEL_WARNING,gSafety.prv.FBK.RemoteControl.StatusID,0,0);
					gSafety.o.State := SAFE_PROGRAM_ERROR;
				ELSE
					//requestMessageToLog(ADR('Acknowledged SK XCHG'), Init_Logbook.pLog, arlogLEVEL_INFO,DEFINE_OFFSET_ERR_START + gSafety.prv.Command_Number,0,0);
					gSafety.o.Status_Print := 'Successfully Acknowledged SK XCHG';
					gSafetyPermInfo.SKey_Exchanged := 1;
					gSafety.o.State := SAFE_PROGRAM_PRINT_STATUS_WAIT;
				END_IF;
			ELSIF gSafety.prv.FBK.RemoteControl.Error THEN
				gSafety.o.Status_Print := 'Error during confirming SK XCHG';
				//requestMessageToLog(ADR('Error during confirming SK XCHG'), Init_Logbook.pLog, arlogLEVEL_WARNING,gSafety.prv.FBK.RemoteControl.StatusID,0,0);
				gSafety.o.State := SAFE_PROGRAM_ERROR;
			ELSIF bgTimerIsTimeOut(gSafety.prv.Timer.Timer_Max_RCTRL_Cmd) THEN
				gSafety.o.Status_Print := 'Timeout confirming SK exchange';
				//requestMessageToLog(ADR('Timeout during SK XCHG confirmation'), Init_Logbook.pLog, arlogLEVEL_WARNING,DEFINE_OFFSET_ERR_START + gSafety.prv.Command_Number,0,0);
				gSafety.o.State := SAFE_PROGRAM_ERROR;
			END_IF;

		SAFE_PROGRAM_CONFIRM_FW:
			gSafety.o.Status_Print := 'Confirming FW mismatch';

			IF gSafety.prv.FBK.RemoteControl.Done AND NOT gSafety.prv.FBK.RemoteControl.Error THEN
				IF gSafety.prv.FBK.RemoteControl.Error THEN
					//requestMessageToLog(ADR('Error during Firmware ACK'), Init_Logbook.pLog, arlogLEVEL_WARNING,gSafety.prv.FBK.RemoteControl.StatusID,0,0);
					gSafety.o.State := SAFE_PROGRAM_ERROR;
				ELSE
					//requestMessageToLog(ADR('Ackd FW'), Init_Logbook.pLog, arlogLEVEL_INFO,DEFINE_OFFSET_ERR_START + gSafety.prv.Command_Number,0,0);
					gSafety.o.Status_Print := 'Successfully acknowledged firmware change';
					gSafety.o.State := SAFE_PROGRAM_PRINT_STATUS_WAIT;
				END_IF;
			ELSIF gSafety.prv.FBK.RemoteControl.Error THEN
				gSafety.o.Status_Print := 'Error Confirming FW mismatch';
				//requestMessageToLog(ADR('Error during Firmware ACK'), Init_Logbook.pLog, arlogLEVEL_WARNING,gSafety.prv.FBK.RemoteControl.StatusID,0,0);
				gSafety.o.State := SAFE_PROGRAM_ERROR;
			ELSIF bgTimerIsTimeOut(gSafety.prv.Timer.Timer_Max_RCTRL_Cmd) THEN
				gSafety.o.Status_Print := 'Timeout acknowledging firmware mismatch';
				//requestMessageToLog(ADR('Timeout during FW ACK'), Init_Logbook.pLog, arlogLEVEL_WARNING,DEFINE_OFFSET_ERR_START + gSafety.prv.Command_Number,0,0);
				gSafety.o.State := SAFE_PROGRAM_ERROR;
			END_IF;

		SAFE_PROGRAM_SCAN:
			gSafety.o.Status_Print := 'Performing System Scan';

			IF gSafety.prv.FBK.RemoteControl.Done AND NOT gSafety.prv.FBK.RemoteControl.Error THEN
				IF gSafety.prv.FBK.RemoteControl.Error THEN
					//requestMessageToLog(ADR('Error during performing system scan'), Init_Logbook.pLog, arlogLEVEL_WARNING,gSafety.prv.FBK.RemoteControl.StatusID,0,0);
					gSafety.o.State := SAFE_PROGRAM_ERROR;
				ELSE
					//requestMessageToLog(ADR('Scanned system'), Init_Logbook.pLog, arlogLEVEL_INFO,DEFINE_OFFSET_ERR_START + gSafety.prv.Command_Number,0,0);
					gSafety.o.Status_Print := 'Successfully Scanned System';
					gSafety.o.State := SAFE_PROGRAM_PRINT_STATUS_WAIT;
				END_IF;
			ELSIF gSafety.prv.FBK.RemoteControl.Error THEN
				gSafety.o.Status_Print := 'Error Performing System Scan';
				//requestMessageToLog(ADR('Error during performing system scan'), Init_Logbook.pLog, arlogLEVEL_WARNING,gSafety.prv.FBK.RemoteControl.StatusID,0,0);
				gSafety.o.State := SAFE_PROGRAM_ERROR;
			ELSIF bgTimerIsTimeOut(gSafety.prv.Timer.Timer_Max_RCTRL_Cmd) THEN
				gSafety.o.Status_Print := 'Timeout during network scan';
				//requestMessageToLog(ADR('Timeout during system scan'), Init_Logbook.pLog, arlogLEVEL_WARNING,DEFINE_OFFSET_ERR_START + gSafety.prv.Command_Number,0,0);
				gSafety.o.State := SAFE_PROGRAM_ERROR;
			END_IF;

		SAFE_PROGRAM_LED_TEST:
			gSafety.o.Status_Print := 'Testing LEDs';

			IF gSafety.prv.FBK.RemoteControl.Done AND NOT gSafety.prv.FBK.RemoteControl.Error THEN
				IF gSafety.prv.FBK.RemoteControl.Error THEN
					//requestMessageToLog(ADR('Error during LED test'), Init_Logbook.pLog, arlogLEVEL_WARNING,gSafety.prv.FBK.RemoteControl.StatusID,0,0);
					gSafety.o.State := SAFE_PROGRAM_ERROR;
				ELSE
					//requestMessageToLog(ADR('LED Test Concluded'), Init_Logbook.pLog, arlogLEVEL_INFO,DEFINE_OFFSET_ERR_START + gSafety.prv.Command_Number,0,0);
					gSafety.o.Status_Print := 'Successfully carried out LED test procedure';
					gSafety.o.State := SAFE_PROGRAM_PRINT_STATUS_WAIT;
				END_IF;
			ELSIF gSafety.prv.FBK.RemoteControl.Error THEN
				gSafety.o.Status_Print := 'Error Testing LEDs';
				//requestMessageToLog(ADR('Error during LED test'), Init_Logbook.pLog, arlogLEVEL_WARNING,gSafety.prv.FBK.RemoteControl.StatusID,0,0);
				gSafety.o.State := SAFE_PROGRAM_ERROR;
			ELSIF bgTimerIsTimeOut(gSafety.prv.Timer.Timer_Max_RCTRL_Cmd) THEN
				gSafety.o.Status_Print := 'Timeout during LED test';
				//requestMessageToLog(ADR('Timeout during LED Test'), Init_Logbook.pLog, arlogLEVEL_WARNING,DEFINE_OFFSET_ERR_START + gSafety.prv.Command_Number,0,0);
				gSafety.o.State := SAFE_PROGRAM_ERROR;
			END_IF;

		SAFE_PROGRAM_CLEAR_DATA:
			gSafety.o.Status_Print := 'Clearing Reloaded Data';

			IF gSafety.prv.FBK.RemoteControl.Done AND NOT gSafety.prv.FBK.RemoteControl.Error THEN
				IF gSafety.prv.FBK.RemoteControl.Error THEN
					//requestMessageToLog(ADR('Error during clear data'), Init_Logbook.pLog, arlogLEVEL_WARNING,gSafety.prv.FBK.RemoteControl.StatusID,0,0);
					gSafety.o.State := SAFE_PROGRAM_ERROR;
				ELSE
					//requestMessageToLog(ADR('Cleared SLX Data'), Init_Logbook.pLog, arlogLEVEL_INFO,DEFINE_OFFSET_ERR_START + gSafety.prv.Command_Number,0,0);
					gSafety.o.Status_Print := 'Successfully cleared SLX data';
					gSafety.o.State := SAFE_PROGRAM_PRINT_STATUS_WAIT;
				END_IF;
			ELSIF gSafety.prv.FBK.RemoteControl.Error THEN
				gSafety.o.Status_Print := 'Error Clearing Reloaded Data';
				//requestMessageToLog(ADR('Error during clear data'), Init_Logbook.pLog, arlogLEVEL_WARNING,gSafety.prv.FBK.RemoteControl.StatusID,0,0);
				gSafety.o.State := SAFE_PROGRAM_ERROR;
			ELSIF bgTimerIsTimeOut(gSafety.prv.Timer.Timer_Max_RCTRL_Cmd) THEN
				gSafety.o.Status_Print := 'Timeout clearing SLX data';
				//requestMessageToLog(ADR('Timeout during clear SLX data'), Init_Logbook.pLog, arlogLEVEL_WARNING,DEFINE_OFFSET_ERR_START + gSafety.prv.Command_Number,0,0);
				gSafety.o.State := SAFE_PROGRAM_ERROR;
			END_IF;

		SAFE_PROGRAM_CONFIRM_MODULES:
			gSafety.o.Status_Print := 'Confirming Module UDID mismatch';

			IF gSafety.prv.FBK.RemoteControl.Done AND NOT gSafety.prv.FBK.RemoteControl.Error THEN
				IF gSafety.prv.FBK.RemoteControl.Error THEN
					//requestMessageToLog(ADR('Error during UDID mismatch confirmation'), Init_Logbook.pLog, arlogLEVEL_WARNING,gSafety.prv.FBK.RemoteControl.StatusID,0,0);
					gSafety.o.State := SAFE_PROGRAM_ERROR;
				ELSE
					//requestMessageToLog(ADR('Ackd UDID mismatch'), Init_Logbook.pLog, arlogLEVEL_INFO,DEFINE_OFFSET_ERR_START + gSafety.prv.Command_Number,0,0);
					gSafety.o.Status_Print := 'Successfully completed UDID mismatch acknowledgement';
					gSafetyPermInfo.ACK_UDID_Firmware := 1;
					gSafety.o.State := SAFE_PROGRAM_PRINT_STATUS_WAIT;
				END_IF;
			ELSIF gSafety.prv.FBK.RemoteControl.Error THEN
				gSafety.o.Status_Print := 'Error Confirming Module UDID mismatch';
				//requestMessageToLog(ADR('Error during UDID mismatch confirmation'), Init_Logbook.pLog, arlogLEVEL_WARNING,gSafety.prv.FBK.RemoteControl.StatusID,0,0);
				gSafety.o.State := SAFE_PROGRAM_ERROR;
			ELSIF bgTimerIsTimeOut(gSafety.prv.Timer.Timer_Max_RCTRL_Cmd) THEN
				gSafety.o.Status_Print := 'Timeout during UDID mismatch acknowledgment';
				//requestMessageToLog(ADR('Timeout during UDID mismatch ACK'), Init_Logbook.pLog, arlogLEVEL_WARNING,DEFINE_OFFSET_ERR_START + gSafety.prv.Command_Number,0,0);
				gSafety.o.State := SAFE_PROGRAM_ERROR;
			END_IF;

		SAFE_PROGRAM_RESET:
			gSafety.o.Status_Print := 'Resetting Data';

			IF gSafety.prv.FBK.RemoteControl.Done AND NOT gSafety.prv.FBK.RemoteControl.Error THEN
				IF gSafety.prv.FBK.RemoteControl.Error THEN
					//requestMessageToLog(ADR('Error during data reset'), Init_Logbook.pLog, arlogLEVEL_WARNING,gSafety.prv.FBK.RemoteControl.StatusID,0,0);
					gSafety.o.State := SAFE_PROGRAM_ERROR;
				ELSE
					//requestMessageToLog(ADR('Reset SLX data'), Init_Logbook.pLog, arlogLEVEL_INFO,DEFINE_OFFSET_ERR_START + gSafety.prv.Command_Number,0,0);
					gSafety.o.Status_Print := 'Successfully reset SLX data';
					gSafety.o.State := SAFE_PROGRAM_PRINT_STATUS_WAIT;
				END_IF;
			ELSIF gSafety.prv.FBK.RemoteControl.Error THEN
				gSafety.o.Status_Print := 'Data Reset Error';
				//requestMessageToLog(ADR('Error during data reset'), Init_Logbook.pLog, arlogLEVEL_WARNING,gSafety.prv.FBK.RemoteControl.StatusID,0,0);
				gSafety.o.State := SAFE_PROGRAM_ERROR;
			ELSIF bgTimerIsTimeOut(gSafety.prv.Timer.Timer_Max_RCTRL_Cmd) THEN
				gSafety.o.Status_Print := 'Timeout resetting SLX';
				//requestMessageToLog(ADR('Timeout during SLX data reset'), Init_Logbook.pLog, arlogLEVEL_WARNING,DEFINE_OFFSET_ERR_START + gSafety.prv.Command_Number,0,0);
				gSafety.o.State := SAFE_PROGRAM_ERROR;
			END_IF;

		SAFE_PROGRAM_ERROR:
			Action_Reset_FBK;
			brsmemset(ADR(gSafety.i.Command), 0, SIZEOF(paiSL_Operations_typ));
			brsmemset(ADR(gSafety.o.Command_Being_Executed), 0, SIZEOF(paiSL_Operations_typ));

			IF bgTimerIsTimeOut(gSafety.prv.Timer.Timer_Error_Retry) THEN
				gSafety.o.Status_Print := 'Returning...';

				bgTimerStart(gSafety.prv.Timer.Timer_Print_HMI_Status, Tms(DEFINE_TIME_PRINT_HMI_STATUS));
				gSafety.o.State := SAFE_PROGRAM_PRINT_STATUS_WAIT;
			END_IF;

		SAFE_PROGRAM_PRINT_STATUS_WAIT:
			Action_Reset_FBK;

			brsmemset(ADR(gSafety.o.Command_Being_Executed), 0, SIZEOF(paiSL_Operations_typ));

			IF bgTimerIsTimeOut(gSafety.prv.Timer.Timer_Print_HMI_Status) THEN

				gSafety.prv.Command_Number := gSafety.prv.Command_Number + 1;
				gSafety.prv.Data.RemoteControlCmd.Number := gSafety.prv.Command_Number;

				bgTimerStart(gSafety.prv.Timer.Timer_Max_RCTRL_Cmd, Tms(DEFINE_TIME_MAX_RCTRL_CMD));
				gSafety.prv.FBK.RemoteControl.Execute := TRUE;
				gSafety.o.State := SAFE_PROGRAM_READ_STATUS;
			END_IF;
	END_CASE;

	gSafety.prv.FBK.RemoteControl();
	gSafety.prv.FBK.DownloadApplication();
	gSafety.prv.FBK.UDID_Low();
	gSafety.prv.FBK.UDID_High();

	bgTimerCyclic(gSafety.prv.Timer.Timer_Print_HMI_Status);
	bgTimerCyclic(gSafety.prv.Timer.Timer_Max_RCTRL_Cmd);
	bgTimerCyclic(gSafety.prv.Timer.Timer_Error_Retry);
	bgTimerCyclic(gSafety.prv.Timer.Timer_Rescan);

	gSafety.o.State_Old := gSafety.o.State;
END_PROGRAM
```

Listed in the project but not available here: Logical/doc, Logical/Alarms.typ, Logical/Enumerations.typ, Logical/ControlStructures.typ, Logical/IO.typ, Logical/varPkg.var, Logical/UserLibraries/wbrServices/bglibasWBR/bglibasWBR.typ, Logical/UserLibraries/wbrServices/bglibasWBR/bglibasWBR.var, Logical/UserLibraries/wbrServices/bglibasWBR/bglibasWBR.fun, Logical/UserLibraries/wbrServices/bglibasWBR/bgssm.c, Logical/UserLibraries/wbrServices/bglibasWBR/bgfifo.c, Logical/UserLibraries/wbrServices/bglibasWBR/bgTimer1ms.c, Logical/UserLibraries/wbrServices/bglibasWBR/wbrFunc.h, Logical/UserLibraries/wbrServices/InitSP/runFirst/runFirstInit.c, Logical/UserLibraries/wbrServices/TimerServices/TimerServices.typ, Logical/UserLibraries/wbrServices/TimerServices/TimerServices.var, Logical/UserLibraries/wbrServices/TimerServices/msTimeSvc, Logical/UserLibraries/wbrServices/wbrListSvc/wbrListSvc.typ, Logical/UserLibraries/wbrServices/wbrListSvc/wbrListSvc.var, Logical/UserLibraries/wbrServices/wbrServices_C_Includes/bglibasWBR_C.h, Logical/UserLibraries/wbrServices/wbrsprintf/cvtflasc.c, Logical/UserLibraries/wbrServices/wbrsprintf/ofmt.c, Logical/UserLibraries/wbrServices/wbrsprintf/wbrsprintf.c, Logical/UserLibraries/wbrServices/wbrSvcUtilities/wbrBytUtil/wbrBytUtil.typ, Logical/UserLibraries/wbrServices/wbrSvcUtilities/wbrBytUtil/wbrBytUtil.fun, Logical/UserLibraries/wbrServices/wbrSvcUtilities/wbrFltUtil/wbrFltUtil.fun, Logical/UserLibraries/wbrServices/wbrSvcUtilities/wbrFltUtil/wbrFloatUtilities.c, Logical/UserLibraries/jgLibs/jgLibC/Constants.var, Logical/Application_Logic/Control, Logical/Application_Logic/FeedRoller, Logical/Application_Logic/lib5200/Belt.typ, Logical/Application_Logic/lib5200/IO.typ, Logical/Application_Logic/lib5200/appGlobal.typ, Logical/Application_Logic/lib5200/VBlocks.typ, Logical/Application_Logic/lib5200/Statistics.typ, Logical/Application_Logic/lib5200/Global_Constants.var, Logical/Application_Logic/lib5200/lib5200.fun, Logical/Application_Logic/pkgInspect/Insp_Global_Var.var, Logical/Application_Logic/pkgInspect/HMITableTexts, Logical/paiComponents/Libraries/sprintf2/cvtflasc.c, Logical/paiComponents/Libraries/sprintf2/ofmt.c, Logical/paiComponents/Libraries/sprintf2/sprintf.c, Logical/paiComponents/Libraries/sprintf2/sprintf2.h, Logical/paiComponents/paiFileService, Logical/paiComponents/paiPing/paiPingService/paiPingService.c, Logical/paiComponents/paiPing/paiPingService/paiPingService.typ, Logical/paiComponents/paiPing/paiPingService/paiPingService.var, Logical/paiComponents/paiPing/paiPingService/paiPing.c, Logical/paiComponents/paiUser/paiUser.typ, Logical/paiComponents/paiUser/paiUser.var, Logical/paiComponents/paiUser/paiUser, Logical/paiComponents/paiUDP/paiUDPService/paiUDPService.typ, Logical/paiComponents/paiUDP/paiUDPService/paiUDPService.var, Logical/paiComponents/paiUDP/paiUDPService/paiUdpserv.c, Logical/paiComponents/paiUDP/paiUDPService/paiUdpclient.c, Logical/paiComponents/paiUDP/paiUDPService/paiUdpService.h, Logical/paiComponents/paiUDP/udpApp/udpApp.c, Logical/paiComponents/paiUDP/paiUDPService/paiUdpclient.c, Logical/paiComponents/paiUDP/paiUDPService/paiUdpserv.c, Logical/paiComponents/bglib/bgstring.c, Logical/paiComponents/bglib/bgringbuffer.c, Logical/paiComponents/paiTemplate/paiHMI/paiConfigSys.typ, Logical/paiComponents/paiTemplate/paiHMI/paiConfig.var, Logical/paiComponents/paiTemplate/paiHMI/paiHMI.var, Logical/paiComponents/paiTemplate/paiHMI/paiHmi, Logical/paiComponents/paiUtility/paiBnRHW.typ, Logical/paiComponents/paiUtility/paiProjectInfo.typ, Logical/HMI/Generic_Controls.typ, Logical/HMI/HMI_Pages.typ, Logical/HMI/HMIdialog.typ, Logical/HMI/HMImsgScroll.typ, Logical/HMI/HMIForceIO.typ, Logical/HMI/HMIalert.typ, Logical/HMI/HMI.typ, Logical/HMI/HMI.var, Logical/HMI/ForceIO, Logical/HMI/HMITableManager, Logical/pkgRecCfg/ParStructs.typ, Logical/pkgRecCfg/RecCfg.var, Logical/pkgAlert/AlarmX/Types.typ, Logical/pkgPVListView/HMITableManager/Main.st, Logical/pkgPVListView/HMITableManager/Types.typ, Logical/FeedAxisobj, Logical/Application/Master/ControlLogic/Main.st, Logical/Application/Master/ControlLogic/Types.typ, Logical/Application/Master/ControlLogic/Variables.var, Logical/Application/Master/ControlLogic/Action_Set_Colorbar_IO.st, Logical/Application/Master/ControlLogic/Action_Manage_Update_Total_Runtime.st, Logical/Application/Master/libAS52XX/Application_Rec_Config.typ, Logical/Application/Master/libAS52XX/libAS52XX.fun, Logical/Application/Master/libAS52XX/FLASH.st, Logical/pkgMpViewAux/MpView_Aux_Global.var, Logical/pkgSafety/Safety_var.var
